Yaskawa INFORM job: DPRINT3D12.JBI

/JOB
//NAME DPRINT3D12
//POS
///NPOS 943,0,0,0,0,0
///TOOL 9
///POSTYPE PULSE
///PULSE
C00000=36380,49514,-121175,76822,-116146,-90921,0
C00001=36311,52030,-113689,77796,-117915,-88696,0
C00002=40966,48656,-123948,71642,-117366,-92253,0
C00003=39960,48244,-125237,72563,-116574,-92522,0
C00004=35348,51596,-114929,78624,-117133,-88953,0
C00005=36233,51994,-113792,77862,-117850,-88717,0
C00006=35618,52329,-112814,78609,-117751,-88361,0
C00007=36492,52745,-111642,77875,-118483,-88119,0
C00008=42195,48620,-124093,70310,-117822,-92440,0
C00009=39827,47660,-127132,72487,-115961,-93077,0
C00010=34247,51723,-114541,79790,-116651,-88720,0
C00011=35148,52115,-113421,79010,-117367,-88487,0
C00012=34913,52339,-112774,79327,-117384,-88271,0
C00013=35382,52553,-112168,78930,-117768,-88145,0
C00014=35564,52380,-112668,78682,-117754,-88312,0
C00015=36124,52085,-113528,78006,-117855,-88627,0
C00016=41195,47951,-126215,71124,-116768,-92950,0
C00017=43098,47003,-129405,68692,-116443,-94111,0
C00018=39318,50776,-117422,74212,-118481,-90143,0
C00019=42795,52637,-112076,71349,-121668,-89077,0
C00020=34867,52594,-112042,79464,-117518,-88051,0
C00021=33535,53991,-108076,81279,-117593,-86746,0
C00022=36088,51585,-114978,77862,-117500,-89049,0
C00023=40156,48632,-124008,72500,-117014,-92178,0
C00024=40156,48569,-124026,72509,-117038,-92154,0
C00025=27110,53258,-109893,66609,-124629,-89161,0
C00026=36380,49453,-121193,76831,-116167,-90898,0
C00027=36311,51973,-113707,77805,-117932,-88673,0
C00028=40967,48594,-123967,71652,-117390,-92229,0
C00029=39960,48181,-125257,72572,-116598,-92498,0
C00030=35348,51539,-114948,78633,-117151,-88931,0
C00031=36233,51937,-113810,77871,-117868,-88695,0
C00032=35619,52272,-112832,78618,-117768,-88339,0
C00033=36492,52688,-111660,77885,-118500,-88098,0
C00034=42195,48557,-124112,70319,-117846,-92417,0
C00035=39828,47596,-127151,72495,-115985,-93052,0
C00036=34247,51665,-114559,79799,-116667,-88698,0
C00037=35149,52058,-113439,79019,-117384,-88465,0
C00038=34914,52282,-112792,79336,-117401,-88249,0
C00039=35382,52497,-112186,78939,-117785,-88123,0
C00040=35565,52323,-112686,78691,-117771,-88290,0
C00041=36125,52027,-113546,78015,-117872,-88605,0
C00042=41195,47887,-126234,71133,-116793,-92926,0
C00043=43079,46945,-129394,68725,-116474,-94076,0
C00044=39319,50717,-117440,74222,-118503,-90120,0
C00045=42764,52562,-112148,71385,-121659,-89066,0
C00046=34867,52538,-112060,79473,-117534,-88029,0
C00047=33548,53922,-108133,81271,-117607,-86737,0
C00048=36088,51527,-114996,77871,-117518,-89026,0
C00049=40156,48569,-124026,72509,-117038,-92154,0
C00050=40157,48507,-124046,72518,-117061,-92130,0
C00051=27147,53215,-109874,66589,-124683,-89138,0
C00052=36381,49392,-121212,76839,-116187,-90874,0
C00053=36312,51915,-113725,77814,-117950,-88651,0
C00054=40967,48531,-123986,71661,-117414,-92206,0
C00055=39961,48118,-125275,72581,-116622,-92474,0
C00056=35348,51481,-114966,78642,-117168,-88908,0
C00057=36234,51879,-113828,77880,-117886,-88673,0
C00058=35619,52216,-112850,78628,-117785,-88317,0
C00059=36492,52632,-111678,77894,-118517,-88076,0
C00060=42195,48495,-124131,70329,-117871,-92394,0
C00061=39828,47531,-127170,72504,-116010,-93028,0
C00062=34248,51608,-114577,79808,-116683,-88676,0
C00063=35149,52001,-113457,79028,-117401,-88442,0
C00064=34914,52225,-112810,79345,-117417,-88227,0
C00065=35382,52440,-112204,78948,-117801,-88101,0
C00066=35565,52266,-112704,78701,-117788,-88268,0
C00067=36125,51970,-113564,78024,-117890,-88583,0
C00068=41196,47823,-126253,71142,-116817,-92902,0
C00069=43061,46888,-129383,68758,-116505,-94040,0
C00070=39319,50658,-117459,74232,-118524,-90097,0
C00071=42733,52486,-112219,71420,-121648,-89055,0
C00072=34868,52481,-112077,79482,-117551,-88007,0
C00073=33561,53853,-108190,81263,-117622,-86728,0
C00074=36088,51469,-115014,77880,-117536,-89004,0
C00075=40157,48507,-124046,72518,-117061,-92130,0
C00076=40157,48444,-124064,72528,-117085,-92106,0
C00077=27184,53173,-109856,66568,-124737,-89114,0
C00078=36381,49332,-121230,76848,-116206,-90851,0
C00079=36312,51858,-113743,77823,-117968,-88629,0
C00080=40968,48469,-124004,71671,-117438,-92182,0
C00081=39961,48055,-125294,72590,-116645,-92450,0
C00082=35349,51423,-114983,78651,-117185,-88885,0
C00083=36234,51822,-113846,77890,-117903,-88650,0
C00084=35619,52159,-112868,78637,-117801,-88295,0
C00085=36493,52576,-111696,77904,-118534,-88054,0
C00086=42196,48432,-124149,70338,-117896,-92370,0
C00087=39828,47467,-127189,72513,-116034,-93003,0
C00088=34248,51550,-114595,79816,-116700,-88653,0
C00089=35150,51944,-113475,79037,-117417,-88420,0
C00090=34914,52168,-112827,79354,-117435,-88204,0
C00091=35383,52383,-112221,78957,-117818,-88079,0
C00092=35565,52209,-112721,78710,-117806,-88246,0
C00093=36125,51913,-113582,78034,-117908,-88561,0
C00094=41196,47759,-126272,71151,-116843,-92878,0
C00095=43042,46831,-129373,68792,-116536,-94005,0
C00096=39320,50599,-117477,74242,-118545,-90075,0
C00097=42701,52411,-112290,71456,-121639,-89045,0
C00098=34868,52424,-112095,79491,-117568,-87985,0
C00099=33573,53785,-108246,81255,-117636,-86720,0
C00100=36089,51411,-115032,77889,-117554,-88982,0
C00101=40157,48444,-124064,72528,-117085,-92106,0
C00102=40157,48382,-124082,72537,-117108,-92083,0
C00103=27222,53130,-109837,66548,-124791,-89091,0
C00104=36381,49271,-121249,76857,-116226,-90827,0
C00105=36312,51801,-113761,77833,-117986,-88607,0
C00106=40968,48407,-124023,71680,-117462,-92159,0
C00107=39962,47992,-125312,72599,-116669,-92426,0
C00108=35349,51365,-115002,78660,-117202,-88863,0
C00109=36234,51765,-113864,77899,-117922,-88628,0
C00110=35620,52102,-112886,78646,-117818,-88272,0
C00111=36493,52519,-111713,77913,-118553,-88032,0
C00112=42196,48370,-124167,70348,-117922,-92347,0
C00113=39829,47402,-127207,72522,-116059,-92979,0
C00114=34248,51492,-114613,79825,-116716,-88631,0
C00115=35150,51887,-113492,79046,-117435,-88398,0
C00116=34915,52111,-112845,79363,-117451,-88182,0
C00117=35383,52327,-112239,78966,-117836,-88057,0
C00118=35566,52153,-112739,78719,-117823,-88224,0
C00119=36126,51856,-113599,78043,-117925,-88538,0
C00120=41196,47695,-126290,71161,-116868,-92854,0
C00121=43024,46774,-129362,68825,-116567,-93970,0
C00122=39320,50540,-117494,74251,-118565,-90053,0
C00123=42670,52335,-112361,71492,-121630,-89034,0
C00124=34868,52368,-112113,79500,-117584,-87963,0
C00125=33586,53716,-108303,81247,-117649,-86710,0
C00126=36089,51353,-115050,77899,-117572,-88959,0
C00127=40157,48382,-124082,72537,-117108,-92083,0
C00128=40158,48319,-124101,72546,-117131,-92059,0
C00129=27259,53088,-109818,66528,-124845,-89067,0
C00130=36382,49210,-121266,76866,-116246,-90804,0
C00131=36313,51744,-113779,77842,-118003,-88585,0
C00132=40968,48344,-124041,71689,-117486,-92135,0
C00133=39962,47928,-125330,72608,-116693,-92402,0
C00134=35350,51307,-115019,78669,-117220,-88840,0
C00135=36235,51707,-113881,77908,-117939,-88606,0
C00136=35620,52045,-112903,78655,-117836,-88250,0
C00137=36493,52463,-111731,77923,-118570,-88010,0
C00138=42197,48307,-124186,70358,-117947,-92323,0
C00139=39829,47338,-127226,72531,-116083,-92955,0
C00140=34248,51435,-114630,79834,-116734,-88608,0
C00141=35150,51830,-113510,79055,-117452,-88375,0
C00142=34915,52055,-112863,79372,-117468,-88160,0
C00143=35383,52270,-112257,78975,-117852,-88035,0
C00144=35566,52096,-112757,78728,-117840,-88201,0
C00145=36126,51799,-113617,78052,-117942,-88516,0
C00146=41197,47632,-126308,71170,-116893,-92830,0
C00147=43005,46717,-129350,68858,-116598,-93934,0
C00148=39320,50481,-117513,74261,-118586,-90030,0
C00149=42639,52260,-112432,71528,-121621,-89023,0
C00150=34868,52311,-112131,79509,-117600,-87941,0
C00151=33599,53647,-108359,81239,-117664,-86702,0
C00152=36089,51296,-115067,77908,-117590,-88936,0
C00153=40158,48319,-124101,72546,-117131,-92059,0
C00154=40158,48257,-124119,72556,-117155,-92035,0
C00155=27296,53046,-109799,66508,-124901,-89043,0
C00156=36382,49149,-121284,76874,-116266,-90780,0
C00157=36313,51687,-113796,77851,-118022,-88563,0
C00158=40969,48282,-124059,71699,-117510,-92111,0
C00159=39963,47865,-125349,72617,-116716,-92378,0
C00160=35350,51250,-115036,78678,-117238,-88817,0
C00161=36235,51650,-113899,77918,-117956,-88584,0
C00162=35620,51988,-112921,78664,-117853,-88228,0
C00163=36494,52407,-111748,77932,-118587,-87988,0
C00164=42197,48245,-124204,70368,-117972,-92300,0
C00165=39830,47274,-127245,72540,-116107,-92930,0
C00166=34249,51377,-114648,79842,-116750,-88585,0
C00167=35150,51773,-113528,79064,-117469,-88353,0
C00168=34915,51998,-112880,79381,-117484,-88137,0
C00169=35384,52214,-112274,78984,-117869,-88013,0
C00170=35566,52039,-112774,78737,-117856,-88179,0
C00171=36126,51742,-113635,78061,-117961,-88494,0
C00172=41197,47568,-126327,71179,-116919,-92806,0
C00173=42987,46660,-129340,68891,-116629,-93899,0
C00174=39321,50422,-117530,74271,-118607,-90007,0
C00175=42608,52184,-112503,71563,-121611,-89012,0
C00176=34869,52255,-112148,79518,-117617,-87919,0
C00177=33612,53578,-108415,81230,-117678,-86693,0
C00178=36090,51238,-115084,77917,-117608,-88914,0
C00179=40158,48257,-124119,72556,-117155,-92035,0
C00180=40159,48194,-124136,72565,-117179,-92011,0
C00181=27333,53003,-109780,66488,-124955,-89020,0
C00182=36383,49088,-121303,76883,-116285,-90756,0
C00183=36313,51629,-113814,77861,-118039,-88540,0
C00184=40969,48219,-124078,71709,-117534,-92087,0
C00185=39963,47802,-125367,72626,-116740,-92354,0
C00186=35350,51192,-115055,78687,-117255,-88795,0
C00187=36235,51593,-113917,77927,-117975,-88561,0
C00188=35621,51931,-112938,78674,-117870,-88206,0
C00189=36494,52350,-111766,77942,-118604,-87967,0
C00190=42198,48182,-124223,70377,-117996,-92276,0
C00191=39830,47209,-127263,72548,-116131,-92905,0
C00192=34249,51320,-114665,79851,-116767,-88563,0
C00193=35151,51716,-113545,79073,-117485,-88331,0
C00194=34916,51941,-112898,79390,-117501,-88115,0
C00195=35384,52157,-112292,78994,-117885,-87990,0
C00196=35567,51982,-112792,78747,-117873,-88157,0
C00197=36127,51685,-113652,78071,-117978,-88472,0
C00198=41198,47504,-126345,71188,-116944,-92782,0
C00199=42968,46603,-129328,68924,-116660,-93863,0
C00200=39321,50364,-117548,74281,-118628,-89985,0
C00201=42577,52108,-112573,71599,-121601,-89001,0
C00202=34869,52199,-112166,79527,-117633,-87896,0
C00203=33624,53509,-108472,81222,-117693,-86684,0
C00204=36090,51180,-115103,77926,-117626,-88891,0
C00205=40159,48194,-124136,72565,-117179,-92011,0
C00206=40159,48132,-124155,72574,-117202,-91987,0
C00207=27370,52961,-109760,66468,-125010,-88996,0
C00208=36383,49027,-121320,76892,-116306,-90732,0
C00209=36314,51572,-113831,77870,-118057,-88518,0
C00210=40970,48157,-124095,71718,-117559,-92063,0
C00211=39963,47739,-125386,72636,-116765,-92330,0
C00212=35351,51134,-115072,78696,-117272,-88772,0
C00213=36236,51536,-113934,77936,-117992,-88539,0
C00214=35621,51875,-112956,78683,-117887,-88184,0
C00215=36494,52294,-111783,77952,-118622,-87945,0
C00216=42198,48120,-124241,70387,-118022,-92253,0
C00217=39831,47145,-127282,72557,-116157,-92880,0
C00218=34250,51262,-114683,79860,-116783,-88540,0
C00219=35151,51659,-113563,79082,-117502,-88308,0
C00220=34916,51884,-112915,79399,-117517,-88093,0
C00221=35384,52101,-112309,79003,-117902,-87968,0
C00222=35567,51926,-112809,78756,-117891,-88135,0
C00223=36127,51628,-113670,78080,-117995,-88449,0
C00224=41198,47440,-126363,71198,-116969,-92758,0
C00225=42950,46547,-129317,68957,-116691,-93828,0
C00226=39321,50305,-117566,74291,-118649,-89962,0
C00227=42546,52033,-112644,71635,-121592,-88990,0
C00228=34869,52142,-112183,79536,-117649,-87874,0
C00229=33637,53440,-108528,81214,-117707,-86675,0
C00230=36090,51122,-115120,77935,-117644,-88869,0
C00231=40159,48132,-124155,72574,-117202,-91987,0
C00232=40160,48070,-124173,72584,-117227,-91964,0
C00233=27407,52919,-109740,66448,-125064,-88972,0
C00234=36383,48966,-121338,76901,-116326,-90708,0
C00235=36314,51515,-113848,77880,-118075,-88495,0
C00236=40970,48095,-124113,71728,-117583,-92040,0
C00237=39964,47676,-125404,72645,-116789,-92305,0
C00238=35351,51077,-115089,78705,-117290,-88749,0
C00239=36236,51479,-113951,77946,-118010,-88517,0
C00240=35621,51818,-112973,78692,-117905,-88161,0
C00241=36495,52238,-111800,77961,-118639,-87923,0
C00242=42198,48057,-124258,70397,-118047,-92229,0
C00243=39831,47081,-127300,72566,-116181,-92856,0
C00244=34250,51205,-114700,79869,-116800,-88517,0
C00245=35151,51602,-113580,79091,-117520,-88286,0
C00246=34916,51828,-112933,79408,-117534,-88071,0
C00247=35385,52044,-112327,79012,-117919,-87946,0
C00248=35567,51869,-112827,78765,-117908,-88112,0
C00249=36127,51570,-113687,78090,-118014,-88427,0
C00250=41198,47377,-126382,71207,-116994,-92734,0
C00251=42932,46490,-129305,68991,-116722,-93793,0
C00252=39322,50246,-117583,74301,-118670,-89940,0
C00253=42514,51957,-112714,71671,-121583,-88979,0
C00254=34870,52086,-112200,79545,-117667,-87852,0
C00255=33650,53371,-108584,81206,-117722,-86666,0
C00256=36091,51065,-115137,77945,-117662,-88846,0
C00257=40160,48070,-124173,72584,-117227,-91964,0
C00258=40160,48007,-124192,72593,-117249,-91940,0
C00259=27444,52877,-109721,66429,-125119,-88948,0
C00260=36384,48906,-121355,76910,-116345,-90684,0
C00261=36314,51458,-113866,77889,-118093,-88473,0
C00262=40970,48032,-124132,71737,-117607,-92016,0
C00263=39964,47613,-125422,72654,-116813,-92281,0
C00264=35351,51019,-115106,78714,-117308,-88727,0
C00265=36236,51421,-113969,77955,-118029,-88494,0
C00266=35622,51761,-112990,78702,-117922,-88139,0
C00267=36495,52182,-111818,77971,-118657,-87901,0
C00268=42199,47995,-124277,70407,-118072,-92206,0
C00269=39831,47016,-127318,72575,-116205,-92831,0
C00270=34250,51147,-114718,79877,-116816,-88494,0
C00271=35152,51545,-113597,79101,-117537,-88263,0
C00272=34917,51771,-112950,79417,-117551,-88049,0
C00273=35385,51988,-112344,79021,-117937,-87924,0
C00274=35568,51812,-112844,78774,-117925,-88090,0
C00275=36128,51513,-113704,78099,-118031,-88405,0
C00276=41199,47313,-126400,71217,-117019,-92709,0
C00277=42913,46433,-129294,69024,-116752,-93757,0
C00278=39322,50187,-117601,74311,-118691,-89917,0
C00279=42483,51882,-112784,71707,-121574,-88968,0
C00280=34870,52029,-112217,79555,-117683,-87830,0
C00281=33663,53302,-108640,81198,-117737,-86657,0
C00282=36091,51007,-115155,77954,-117680,-88823,0
C00283=40160,48007,-124192,72593,-117249,-91940,0
C00284=40160,47945,-124209,72603,-117274,-91915,0
C00285=27481,52836,-109701,66409,-125173,-88925,0
C00286=36384,48845,-121373,76918,-116366,-90660,0
C00287=36315,51401,-113883,77899,-118110,-88451,0
C00288=40971,47970,-124149,71747,-117631,-91992,0
C00289=39965,47549,-125440,72663,-116837,-92257,0
C00290=35351,50961,-115124,78723,-117325,-88704,0
C00291=36237,51364,-113986,77965,-118046,-88472,0
C00292=35622,51704,-113007,78711,-117939,-88117,0
C00293=36495,52125,-111835,77981,-118674,-87878,0
C00294=42199,47932,-124294,70417,-118098,-92182,0
C00295=39832,46952,-127336,72584,-116230,-92807,0
C00296=34250,51090,-114735,79886,-116833,-88472,0
C00297=35152,51488,-113614,79110,-117554,-88241,0
C00298=34917,51714,-112967,79427,-117568,-88026,0
C00299=35385,51931,-112361,79031,-117953,-87902,0
C00300=35568,51756,-112861,78784,-117942,-88068,0
C00301=36128,51456,-113721,78108,-118049,-88382,0
C00302=41199,47249,-126419,71226,-117044,-92685,0
C00303=42895,46377,-129281,69057,-116783,-93721,0
C00304=39323,50128,-117618,74321,-118711,-89894,0
C00305=42452,51806,-112855,71744,-121563,-88957,0
C00306=34870,51973,-112235,79564,-117700,-87807,0
C00307=33675,53233,-108696,81190,-117751,-86648,0
C00308=36091,50949,-115172,77963,-117698,-88801,0
C00309=40160,47945,-124209,72603,-117274,-91915,0
C00310=40161,47882,-124227,72612,-117298,-91892,0
C00311=27518,52794,-109681,66389,-125228,-88901,0
C00312=36384,48784,-121391,76927,-116385,-90636,0
C00313=36315,51344,-113900,77908,-118129,-88428,0
C00314=40971,47908,-124167,71757,-117655,-91968,0
C00315=39965,47486,-125458,72673,-116860,-92233,0
C00316=35352,50904,-115141,78732,-117343,-88682,0
C00317=36237,51307,-114003,77974,-118064,-88449,0
C00318=35622,51648,-113025,78720,-117956,-88094,0
C00319=36496,52069,-111852,77990,-118692,-87856,0
C00320=42200,47870,-124312,70427,-118123,-92158,0
C00321=39832,46888,-127354,72593,-116254,-92782,0
C00322=34251,51032,-114752,79895,-116850,-88449,0
C00323=35152,51431,-113631,79119,-117570,-88219,0
C00324=34917,51658,-112984,79436,-117584,-88003,0
C00325=35386,51875,-112378,79040,-117970,-87880,0
C00326=35568,51699,-112878,78793,-117960,-88046,0
C00327=36128,51399,-113738,78118,-118067,-88360,0
C00328=41200,47185,-126436,71235,-117069,-92660,0
C00329=42876,46320,-129270,69091,-116814,-93685,0
C00330=39323,50069,-117636,74331,-118733,-89871,0
C00331=42420,51731,-112925,71780,-121554,-88945,0
C00332=34871,51916,-112252,79573,-117716,-87785,0
C00333=33688,53165,-108751,81182,-117765,-86638,0
C00334=36092,50892,-115189,77973,-117716,-88778,0
C00335=40161,47882,-124227,72612,-117298,-91892,0
C00336=40161,47820,-124244,72622,-117321,-91868,0
C00337=27555,52752,-109661,66370,-125283,-88877,0
C00338=36385,48723,-121408,76936,-116406,-90612,0
C00339=36315,51287,-113917,77918,-118147,-88406,0
C00340=40972,47845,-124185,71766,-117679,-91944,0
C00341=39965,47423,-125475,72682,-116884,-92208,0
C00342=35352,50846,-115158,78741,-117360,-88658,0
C00343=36237,51250,-114020,77984,-118081,-88427,0
C00344=35623,51591,-113041,78730,-117973,-88072,0
C00345=36496,52013,-111869,78000,-118709,-87834,0
C00346=42200,47807,-124329,70437,-118148,-92134,0
C00347=39833,46824,-127372,72602,-116278,-92757,0
C00348=34251,50975,-114769,79904,-116867,-88426,0
C00349=35153,51374,-113648,79128,-117587,-88196,0
C00350=34918,51601,-113001,79445,-117601,-87981,0
C00351=35386,51819,-112395,79049,-117987,-87857,0
C00352=35569,51643,-112895,78803,-117977,-88023,0
C00353=36129,51342,-113755,78127,-118085,-88337,0
C00354=41200,47122,-126454,71245,-117096,-92636,0
C00355=42858,46264,-129258,69124,-116845,-93650,0
C00356=39323,50011,-117653,74341,-118754,-89848,0
C00357=42389,51655,-112995,71816,-121545,-88934,0
C00358=34871,51860,-112269,79582,-117732,-87762,0
C00359=33701,53096,-108807,81174,-117780,-86629,0
C00360=36092,50834,-115206,77982,-117734,-88755,0
C00361=40161,47820,-124244,72622,-117321,-91868,0
C00362=40162,47758,-124262,72631,-117345,-91843,0
C00363=27592,52710,-109641,66351,-125337,-88853,0
C00364=36385,48663,-121426,76945,-116426,-90588,0
C00365=36316,51230,-113934,77927,-118164,-88383,0
C00366=40972,47783,-124202,71776,-117705,-91921,0
C00367=39966,47360,-125494,72692,-116908,-92184,0
C00368=35352,50788,-115175,78750,-117378,-88636,0
C00369=36238,51193,-114037,77993,-118100,-88404,0
C00370=35623,51534,-113058,78739,-117991,-88050,0
C00371=36496,51957,-111886,78010,-118727,-87812,0
C00372=42201,47745,-124348,70447,-118173,-92110,0
C00373=39833,46759,-127390,72612,-116304,-92732,0
C00374=34251,50917,-114786,79913,-116883,-88403,0
C00375=35153,51317,-113665,79137,-117605,-88173,0
C00376=34918,51544,-113018,79454,-117618,-87959,0
C00377=35386,51762,-112412,79059,-118003,-87835,0
C00378=35569,51586,-112912,78812,-117994,-88001,0
C00379=36129,51286,-113772,78137,-118102,-88315,0
C00380=41201,47058,-126471,71254,-117121,-92612,0
C00381=42840,46207,-129246,69157,-116875,-93614,0
C00382=39324,49952,-117670,74351,-118774,-89825,0
C00383=42357,51579,-113064,71852,-121536,-88922,0
C00384=34871,51804,-112285,79592,-117749,-87740,0
C00385=33714,53027,-108862,81166,-117795,-86620,0
C00386=36093,50776,-115224,77992,-117753,-88733,0
C00387=40162,47758,-124262,72631,-117345,-91843,0
C00388=40162,47695,-124280,72641,-117369,-91820,0
C00389=27629,52669,-109620,66331,-125392,-88830,0
C00390=36385,48602,-121443,76954,-116445,-90565,0
C00391=36316,51173,-113951,77937,-118183,-88361,0
C00392=40972,47721,-124220,71786,-117729,-91897,0
C00393=39966,47297,-125511,72701,-116932,-92160,0
C00394=35353,50731,-115191,78760,-117395,-88613,0
C00395=36238,51136,-114054,78003,-118117,-88382,0
C00396=35623,51478,-113075,78749,-118008,-88027,0
C00397=36497,51901,-111902,78020,-118745,-87790,0
C00398=42201,47683,-124365,70457,-118199,-92087,0
C00399=39833,46695,-127408,72621,-116328,-92707,0
C00400=34252,50860,-114803,79922,-116900,-88380,0
C00401=35153,51260,-113682,79147,-117622,-88151,0
C00402=34918,51488,-113035,79463,-117634,-87936,0
C00403=35387,51706,-112429,79068,-118021,-87812,0
C00404=35569,51529,-112929,78821,-118011,-87978,0
C00405=36129,51229,-113789,78146,-118121,-88292,0
C00406=41201,46995,-126490,71264,-117146,-92587,0
C00407=42821,46151,-129234,69191,-116906,-93578,0
C00408=39324,49893,-117686,74361,-118796,-89803,0
C00409=42326,51504,-113134,71889,-121527,-88911,0
C00410=34872,51748,-112302,79601,-117765,-87718,0
C00411=33726,52958,-108918,81158,-117809,-86611,0
C00412=36093,50719,-115241,78001,-117770,-88709,0
C00413=40162,47695,-124280,72641,-117369,-91820,0
C00414=40162,47633,-124297,72651,-117392,-91795,0
C00415=27666,52627,-109600,66312,-125448,-88806,0
C00416=36386,48541,-121460,76963,-116466,-90540,0
C00417=36316,51116,-113968,77946,-118200,-88338,0
C00418=40973,47658,-124238,71796,-117753,-91872,0
C00419=39967,47234,-125528,72710,-116956,-92135,0
C00420=35353,50673,-115209,78769,-117413,-88590,0
C00421=36238,51079,-114071,78012,-118135,-88359,0
C00422=35624,51421,-113092,78758,-118025,-88004,0
C00423=36497,51845,-111919,78030,-118762,-87768,0
C00424=42201,47620,-124382,70467,-118224,-92063,0
C00425=39834,46631,-127425,72630,-116353,-92683,0
C00426=34252,50803,-114820,79931,-116917,-88357,0
C00427=35154,51203,-113699,79156,-117639,-88128,0
C00428=34919,51431,-113052,79473,-117652,-87913,0
C00429=35387,51650,-112445,79078,-118038,-87790,0
C00430=35570,51473,-112945,78831,-118029,-87956,0
C00431=36130,51172,-113806,78156,-118138,-88270,0
C00432=41201,46931,-126507,71274,-117171,-92563,0
C00433=42803,46095,-129221,69224,-116937,-93542,0
C00434=39324,49834,-117703,74371,-118817,-89779,0
C00435=42294,51428,-113203,71925,-121517,-88899,0
C00436=34872,51691,-112319,79610,-117783,-87696,0
C00437=33739,52889,-108973,81150,-117824,-86601,0
C00438=36093,50661,-115257,78010,-117788,-88687,0
C00439=40162,47633,-124297,72651,-117392,-91795,0
C00440=40163,47571,-124314,72660,-117416,-91771,0
C00441=27702,52586,-109579,66293,-125503,-88781,0
C00442=36386,48481,-121477,76972,-116485,-90516,0
C00443=36317,51059,-113984,77956,-118218,-88315,0
C00444=40973,47596,-124255,71806,-117777,-91849,0
C00445=39967,47171,-125546,72720,-116981,-92110,0
C00446=35353,50616,-115226,78778,-117431,-88567,0
C00447=36239,51022,-114087,78022,-118154,-88336,0
C00448=35624,51365,-113109,78767,-118042,-87982,0
C00449=36497,51789,-111936,78039,-118780,-87746,0
C00450=42202,47558,-124400,70477,-118250,-92039,0
C00451=39834,46567,-127444,72639,-116377,-92658,0
C00452=34252,50745,-114836,79940,-116933,-88334,0
C00453=35154,51146,-113716,79165,-117656,-88105,0
C00454=34919,51374,-113068,79482,-117669,-87891,0
C00455=35387,51593,-112462,79087,-118055,-87768,0
C00456=35570,51416,-112962,78840,-118046,-87934,0
C00457=36130,51115,-113823,78166,-118156,-88247,0
C00458=41202,46867,-126524,71283,-117197,-92539,0
C00459=42785,46039,-129209,69258,-116967,-93506,0
C00460=39325,49776,-117721,74381,-118838,-89757,0
C00461=42263,51353,-113273,71962,-121508,-88888,0
C00462=34872,51635,-112336,79619,-117799,-87673,0
C00463=33752,52820,-109028,81142,-117839,-86592,0
C00464=36094,50604,-115274,78020,-117807,-88664,0
C00465=40163,47571,-124314,72660,-117416,-91771,0
C00466=40163,47509,-124332,72670,-117440,-91747,0
C00467=27739,52545,-109558,66274,-125558,-88758,0
C00468=36387,48420,-121494,76981,-116506,-90492,0
C00469=36317,51002,-114001,77966,-118237,-88293,0
C00470=40974,47534,-124272,71816,-117802,-91824,0
C00471=39967,47108,-125564,72729,-117005,-92086,0
C00472=35354,50558,-115242,78787,-117448,-88544,0
C00473=36239,50965,-114104,78032,-118171,-88314,0
C00474=35624,51308,-113125,78777,-118060,-87960,0
C00475=36498,51733,-111952,78049,-118797,-87724,0
C00476=42202,47496,-124417,70487,-118276,-92015,0
C00477=39835,46503,-127461,72648,-116403,-92633,0
C00478=34253,50688,-114853,79948,-116951,-88311,0
C00479=35154,51090,-113732,79175,-117674,-88083,0
C00480=34919,51318,-113085,79491,-117685,-87868,0
C00481=35388,51537,-112478,79097,-118072,-87745,0
C00482=35570,51360,-112979,78850,-118063,-87911,0
C00483=36130,51058,-113839,78175,-118173,-88224,0
C00484=41202,46804,-126543,71293,-117222,-92514,0
C00485=42766,45983,-129196,69291,-116998,-93471,0
C00486=39325,49717,-117737,74392,-118859,-89734,0
C00487=42232,51277,-113342,71998,-121499,-88876,0
C00488=34873,51579,-112352,79629,-117816,-87650,0
C00489=33765,52751,-109083,81134,-117854,-86583,0
C00490=36094,50546,-115290,78029,-117825,-88641,0
C00491=40163,47509,-124332,72670,-117440,-91747,0
C00492=40164,47446,-124349,72680,-117464,-91723,0
C00493=27776,52503,-109537,66255,-125613,-88734,0
C00494=36387,48359,-121512,76990,-116526,-90468,0
C00495=36317,50945,-114017,77975,-118254,-88270,0
C00496=40974,47472,-124289,71826,-117826,-91801,0
C00497=39968,47045,-125581,72739,-117029,-92062,0
C00498=35354,50501,-115259,78797,-117467,-88521,0
C00499=36239,50908,-114120,78041,-118189,-88291,0
C00500=35625,51252,-113142,78787,-118077,-87937,0
C00501=36498,51677,-111969,78059,-118815,-87701,0
C00502=42203,47434,-124434,70497,-118301,-91991,0
C00503=39835,46439,-127478,72658,-116427,-92607,0
C00504=34253,50631,-114870,79958,-116968,-88288,0
C00505=35155,51033,-113749,79184,-117691,-88060,0
C00506=34920,51261,-113101,79501,-117702,-87845,0
C00507=35388,51481,-112495,79106,-118088,-87723,0
C00508=35570,51303,-112995,78859,-118080,-87888,0
C00509=36131,51001,-113856,78185,-118192,-88202,0
C00510=41203,46740,-126560,71303,-117247,-92489,0
C00511=42748,45927,-129183,69325,-117028,-93435,0
C00512=39325,49658,-117754,74402,-118880,-89710,0
C00513=42200,51202,-113411,72035,-121490,-88864,0
C00514=34873,51523,-112369,79638,-117832,-87628,0
C00515=33778,52683,-109139,81126,-117869,-86573,0
C00516=36094,50489,-115307,78039,-117844,-88618,0
C00517=40164,47446,-124349,72680,-117464,-91723,0
C00518=40164,47384,-124366,72690,-117487,-91698,0
C00519=27813,52462,-109516,66237,-125668,-88710,0
C00520=36387,48299,-121528,77000,-116546,-90444,0
C00521=36318,50888,-114034,77985,-118272,-88248,0
C00522=40975,47410,-124306,71836,-117850,-91776,0
C00523=39968,46982,-125598,72749,-117053,-92037,0
C00524=35355,50443,-115275,78806,-117484,-88498,0
C00525=36240,50851,-114137,78051,-118208,-88268,0
C00526=35625,51195,-113158,78796,-118094,-87914,0
C00527=36498,51621,-111985,78069,-118833,-87679,0
C00528=42203,47371,-124451,70507,-118326,-91968,0
C00529=39836,46374,-127495,72667,-116452,-92582,0
C00530=34253,50573,-114886,79967,-116984,-88265,0
C00531=35155,50976,-113765,79193,-117708,-88037,0
C00532=34920,51205,-113118,79510,-117719,-87823,0
C00533=35388,51425,-112511,79116,-118106,-87700,0
C00534=35571,51247,-113012,78869,-118098,-87866,0
C00535=36131,50944,-113872,78195,-118209,-88179,0
C00536=41203,46677,-126577,71312,-117272,-92465,0
C00537=42730,45870,-129171,69358,-117059,-93399,0
C00538=39326,49600,-117770,74412,-118902,-89688,0
C00539=42168,51126,-113480,72071,-121481,-88852,0
C00540=34873,51467,-112385,79648,-117849,-87606,0
C00541=33790,52614,-109194,81119,-117884,-86564,0
C00542=36095,50431,-115324,78049,-117862,-88595,0
C00543=40164,47384,-124366,72690,-117487,-91698,0
C00544=40164,47322,-124382,72699,-117511,-91674,0
C00545=27850,52421,-109495,66218,-125723,-88686,0
C00546=36388,48238,-121545,77009,-116566,-90419,0
C00547=36318,50831,-114050,77995,-118291,-88225,0
C00548=40975,47348,-124324,71846,-117876,-91752,0
C00549=39969,46919,-125615,72758,-117077,-92012,0
C00550=35355,50386,-115291,78816,-117501,-88475,0
C00551=36240,50794,-114153,78061,-118225,-88245,0
C00552=35625,51139,-113174,78806,-118113,-87892,0
C00553=36499,51565,-112001,78079,-118850,-87656,0
C00554=42204,47309,-124468,70518,-118352,-91943,0
C00555=39836,46310,-127513,72676,-116476,-92557,0
C00556=34254,50516,-114903,79976,-117001,-88242,0
C00557=35155,50919,-113782,79203,-117725,-88014,0
C00558=34920,51148,-113134,79519,-117736,-87800,0
C00559=35389,51368,-112528,79125,-118123,-87678,0
C00560=35571,51191,-113028,78879,-118115,-87843,0
C00561=36131,50887,-113889,78204,-118227,-88156,0
C00562=41204,46613,-126594,71322,-117299,-92440,0
C00563=42712,45814,-129158,69392,-117089,-93363,0
C00564=39326,49541,-117787,74422,-118923,-89665,0
C00565=42137,51051,-113549,72108,-121471,-88841,0
C00566=34874,51410,-112401,79657,-117865,-87583,0
C00567=33803,52545,-109248,81111,-117899,-86554,0
C00568=36095,50374,-115340,78058,-117879,-88572,0
C00569=40164,47322,-124382,72699,-117511,-91674,0
C00570=40165,47260,-124400,72709,-117536,-91650,0
C00571=27886,52380,-109474,66199,-125779,-88662,0
C00572=36388,48178,-121561,77018,-116586,-90395,0
C00573=36318,50774,-114067,78005,-118309,-88202,0
C00574=40975,47285,-124340,71856,-117900,-91728,0
C00575=39969,46856,-125631,72768,-117101,-91987,0
C00576=35355,50328,-115309,78825,-117520,-88452,0
C00577=36240,50737,-114170,78070,-118244,-88223,0
C00578=35626,51082,-113191,78815,-118130,-87869,0
C00579=36499,51509,-112018,78089,-118868,-87634,0
C00580=42204,47247,-124486,70528,-118377,-91919,0
C00581=39836,46246,-127530,72686,-116501,-92532,0
C00582=34254,50459,-114919,79985,-117019,-88219,0
C00583=35156,50862,-113798,79212,-117742,-87992,0
C00584=34920,51092,-113150,79529,-117753,-87778,0
C00585=35389,51312,-112544,79135,-118140,-87655,0
C00586=35572,51134,-113044,78888,-118132,-87820,0
C00587=36132,50831,-113905,78214,-118245,-88134,0
C00588=41204,46550,-126612,71332,-117324,-92416,0
C00589=42693,45759,-129146,69425,-117120,-93327,0
C00590=39327,49482,-117803,74433,-118944,-89641,0
C00591=42105,50975,-113617,72145,-121462,-88828,0
C00592=34874,51354,-112418,79666,-117883,-87560,0
C00593=33816,52476,-109303,81103,-117914,-86544,0
C00594=36095,50316,-115357,78068,-117898,-88549,0
C00595=40165,47260,-124400,72709,-117536,-91650,0
C00596=40165,47198,-124417,72719,-117560,-91625,0
C00597=27923,52339,-109452,66181,-125835,-88638,0
C00598=36388,48117,-121578,77027,-116607,-90371,0
C00599=36319,50718,-114083,78015,-118326,-88179,0
C00600=40976,47223,-124357,71866,-117924,-91704,0
C00601=39969,46794,-125649,72778,-117125,-91963,0
C00602=35355,50271,-115325,78834,-117537,-88429,0
C00603=36241,50680,-114186,78080,-118262,-88200,0
C00604=35626,51026,-113207,78825,-118147,-87847,0
C00605=36499,51453,-112034,78099,-118886,-87612,0
C00606=42204,47185,-124502,70538,-118403,-91896,0
C00607=39837,46182,-127547,72695,-116527,-92507,0
C00608=34254,50402,-114935,79994,-117035,-88196,0
C00609=35156,50806,-113814,79222,-117760,-87968,0
C00610=34921,51036,-113166,79538,-117770,-87755,0
C00611=35389,51256,-112560,79145,-118157,-87632,0
C00612=35572,51078,-113060,78898,-118149,-87798,0
C00613=36132,50774,-113921,78224,-118263,-88111,0
C00614=41204,46486,-126629,71342,-117349,-92391,0
C00615=42675,45703,-129133,69459,-117150,-93291,0
C00616=39327,49424,-117819,74443,-118965,-89618,0
C00617=42073,50899,-113686,72182,-121453,-88817,0
C00618=34874,51298,-112434,79676,-117899,-87538,0
C00619=33829,52407,-109358,81095,-117929,-86535,0
C00620=36096,50259,-115373,78077,-117916,-88526,0
C00621=40165,47198,-124417,72719,-117560,-91625,0
C00622=40166,47136,-124433,72729,-117584,-91601,0
C00623=27960,52298,-109431,66163,-125890,-88614,0
C00624=36389,48057,-121594,77036,-116627,-90346,0
C00625=36319,50661,-114099,78024,-118345,-88156,0
C00626=40976,47161,-124373,71876,-117949,-91679,0
C00627=39970,46731,-125666,72787,-117151,-91938,0
C00628=35356,50214,-115341,78844,-117555,-88405,0
C00629=36241,50624,-114202,78090,-118280,-88177,0
C00630=35626,50969,-113223,78835,-118164,-87823,0
C00631=36500,51397,-112050,78109,-118903,-87589,0
C00632=42205,47122,-124519,70548,-118429,-91871,0
C00633=39837,46118,-127564,72705,-116551,-92482,0
C00634=34255,50344,-114951,80003,-117052,-88173,0
C00635=35156,50749,-113830,79231,-117777,-87946,0
C00636=34921,50979,-113183,79548,-117786,-87732,0
C00637=35390,51200,-112576,79154,-118175,-87610,0
C00638=35572,51022,-113076,78908,-118167,-87775,0
C00639=36132,50717,-113937,78234,-118280,-88088,0
C00640=41205,46423,-126645,71352,-117375,-92366,0
C00641=42657,45647,-129119,69492,-117181,-93255,0
C00642=39327,49365,-117837,74453,-118986,-89595,0
C00643=42042,50824,-113754,72218,-121445,-88805,0
C00644=34875,51242,-112450,79685,-117916,-87515,0
C00645=33842,52338,-109412,81087,-117944,-86525,0
C00646=36096,50201,-115389,78087,-117934,-88503,0
C00647=40166,47136,-124433,72729,-117584,-91601,0
C00648=40166,47073,-124450,72739,-117608,-91577,0
C00649=27996,52257,-109409,66144,-125945,-88590,0
C00650=36389,47996,-121612,77046,-116647,-90322,0
C00651=36319,50604,-114115,78034,-118363,-88133,0
C00652=40977,47099,-124390,71886,-117973,-91655,0
C00653=39970,46668,-125683,72797,-117175,-91914,0
C00654=35356,50156,-115357,78853,-117572,-88382,0
C00655=36241,50567,-114218,78100,-118298,-88154,0
C00656=35626,50913,-113239,78844,-118181,-87801,0
C00657=36500,51341,-112066,78119,-118920,-87567,0
C00658=42205,47060,-124535,70559,-118454,-91848,0
C00659=39838,46054,-127582,72714,-116576,-92456,0
C00660=34255,50287,-114967,80012,-117069,-88149,0
C00661=35157,50692,-113846,79241,-117794,-87923,0
C00662=34921,50923,-113198,79557,-117803,-87709,0
C00663=35390,51144,-112592,79164,-118191,-87587,0
C00664=35572,50965,-113092,78917,-118184,-87753,0
C00665=36133,50660,-113953,78243,-118299,-88065,0
C00666=41205,46359,-126662,71361,-117401,-92341,0
C00667=42639,45591,-129106,69526,-117210,-93219,0
C00668=39328,49307,-117853,74464,-119008,-89572,0
C00669=42010,50748,-113823,72255,-121436,-88792,0
C00670=34875,51186,-112466,79695,-117932,-87493,0
C00671=33855,52269,-109467,81079,-117959,-86515,0
C00672=36096,50144,-115405,78097,-117953,-88480,0
C00673=40166,47073,-124450,72739,-117608,-91577,0
C00674=40167,47011,-124466,72749,-117632,-91552,0
C00675=28033,52216,-109387,66126,-126001,-88566,0
C00676=36389,47936,-121628,77055,-116667,-90298,0
C00677=36320,50547,-114131,78044,-118381,-88111,0
C00678=40977,47037,-124406,71896,-117999,-91631,0
C00679=39971,46605,-125699,72807,-117199,-91889,0
C00680=35356,50099,-115373,78863,-117591,-88359,0
C00681=36242,50510,-114234,78110,-118316,-88131,0
C00682=35627,50857,-113255,78854,-118199,-87778,0
C00683=36500,51285,-112082,78129,-118939,-87544,0
C00684=42206,46998,-124552,70569,-118479,-91823,0
C00685=39838,45990,-127599,72724,-116600,-92431,0
C00686=34255,50230,-114983,80021,-117085,-88126,0
C00687=35157,50636,-113862,79250,-117811,-87900,0
C00688=34922,50866,-113214,79566,-117821,-87686,0
C00689=35390,51088,-112608,79174,-118208,-87565,0
C00690=35573,50909,-113108,78927,-118201,-87729,0
C00691=36133,50604,-113969,78253,-118317,-88042,0
C00692=41206,46296,-126679,71371,-117426,-92316,0
C00693=42621,45536,-129093,69560,-117241,-93183,0
C00694=39328,49248,-117869,74474,-119028,-89548,0
C00695=41978,50673,-113891,72292,-121427,-88780,0
C00696=34875,51130,-112482,79704,-117949,-87470,0
C00697=33867,52201,-109521,81072,-117975,-86506,0
C00698=36097,50087,-115421,78106,-117971,-88456,0
C00699=40167,47011,-124466,72749,-117632,-91552,0
C00700=40167,46949,-124483,72759,-117656,-91527,0
C00701=28070,52176,-109365,66108,-126057,-88542,0
C00702=36390,47875,-121644,77064,-116688,-90273,0
C00703=36320,50490,-114147,78054,-118399,-88088,0
C00704=40977,46975,-124424,71906,-118023,-91607,0
C00705=39971,46542,-125716,72816,-117223,-91864,0
C00706=35357,50042,-115389,78872,-117608,-88336,0
C00707=36242,50453,-114250,78120,-118334,-88108,0
C00708=35627,50800,-113271,78864,-118216,-87755,0
C00709=36501,51229,-112097,78139,-118956,-87522,0
C00710=42206,46936,-124568,70580,-118506,-91799,0
C00711=39838,45926,-127615,72733,-116625,-92406,0
C00712=34256,50173,-114999,80030,-117102,-88102,0
C00713=35157,50579,-113878,79260,-117829,-87877,0
C00714=34922,50810,-113230,79576,-117838,-87663,0
C00715=35390,51032,-112624,79183,-118225,-87542,0
C00716=35573,50853,-113124,78937,-118218,-87707,0
C00717=36133,50547,-113985,78263,-118334,-88019,0
C00718=41206,46232,-126696,71381,-117452,-92292,0
C00719=42602,45480,-129079,69593,-117271,-93147,0
C00720=39328,49190,-117885,74485,-119050,-89525,0
C00721=41946,50597,-113959,72329,-121417,-88768,0
C00722=34875,51074,-112498,79714,-117965,-87447,0
C00723=33880,52132,-109576,81064,-117990,-86496,0
C00724=36097,50029,-115437,78116,-117990,-88433,0
C00725=40167,46949,-124483,72759,-117656,-91527,0
C00726=40167,46887,-124500,72769,-117679,-91503,0
C00727=28106,52135,-109343,66090,-126112,-88518,0
C00728=36390,47815,-121660,77074,-116708,-90249,0
C00729=36320,50434,-114163,78064,-118417,-88065,0
C00730=40978,46913,-124440,71916,-118047,-91582,0
C00731=39972,46479,-125733,72826,-117247,-91839,0
C00732=35357,49984,-115404,78882,-117626,-88313,0
C00733=36242,50396,-114266,78129,-118353,-88085,0
C00734=35628,50744,-113287,78874,-118234,-87732,0
C00735=36501,51173,-112113,78149,-118974,-87499,0
C00736=42206,46874,-124585,70590,-118531,-91775,0
C00737=39839,45862,-127632,72743,-116651,-92381,0
C00738=34256,50116,-115016,80040,-117120,-88079,0
C00739=35158,50523,-113894,79269,-117846,-87854,0
C00740=34922,50754,-113246,79586,-117854,-87641,0
C00741=35391,50976,-112640,79193,-118242,-87519,0
C00742=35573,50796,-113140,78947,-118235,-87684,0
C00743=36134,50490,-114001,78273,-118353,-87996,0
C00744=41207,46169,-126713,71391,-117478,-92267,0
C00745=42584,45425,-129065,69627,-117301,-93111,0
C00746=39329,49131,-117901,74495,-119072,-89502,0
C00747=41914,50522,-114027,72366,-121408,-88755,0
C00748=34876,51018,-112513,79723,-117983,-87424,0
C00749=33893,52063,-109630,81056,-118004,-86486,0
C00750=36097,49972,-115452,78126,-118008,-88410,0
C00751=40167,46887,-124500,72769,-117679,-91503,0
C00752=40168,46825,-124516,72779,-117703,-91478,0
C00753=28143,52095,-109320,66072,-126168,-88494,0
C00754=36391,47754,-121676,77083,-116728,-90225,0
C00755=36321,50377,-114178,78074,-118435,-88042,0
C00756=40978,46851,-124456,71927,-118072,-91558,0
C00757=39972,46417,-125749,72836,-117271,-91814,0
C00758=35357,49927,-115420,78891,-117644,-88289,0
C00759=36243,50340,-114281,78139,-118370,-88062,0
C00760=35628,50687,-113302,78883,-118252,-87710,0
C00761=36501,51118,-112129,78160,-118992,-87476,0
C00762=42207,46812,-124602,70601,-118556,-91751,0
C00763=39839,45798,-127648,72752,-116676,-92355,0
C00764=34256,50059,-115030,80049,-117137,-88056,0
C00765=35158,50466,-113910,79279,-117863,-87831,0
C00766=34923,50698,-113262,79595,-117871,-87617,0
C00767=35391,50920,-112655,79203,-118260,-87496,0
C00768=35574,50740,-113156,78956,-118254,-87661,0
C00769=36134,50434,-114017,78283,-118371,-87974,0
C00770=41207,46105,-126729,71401,-117503,-92242,0
C00771=42566,45369,-129052,69661,-117331,-93075,0
C00772=39329,49073,-117917,74506,-119093,-89479,0
C00773=41882,50446,-114095,72404,-121400,-88743,0
C00774=34876,50962,-112529,79733,-118000,-87402,0
C00775=33906,51994,-109684,81048,-118021,-86476,0
C00776=36098,49915,-115468,78136,-118026,-88387,0
C00777=40168,46825,-124516,72779,-117703,-91478,0
C00778=40168,46763,-124532,72789,-117728,-91454,0
C00779=28179,52054,-109298,66054,-126224,-88470,0
C00780=36391,47694,-121692,77092,-116748,-90200,0
C00781=36321,50320,-114194,78084,-118454,-88019,0
C00782=40979,46789,-124472,71937,-118096,-91533,0
C00783=39972,46354,-125765,72846,-117297,-91789,0
C00784=35358,49870,-115436,78901,-117662,-88266,0
C00785=36243,50283,-114297,78149,-118388,-88039,0
C00786=35628,50631,-113318,78893,-118269,-87686,0
C00787=36502,51062,-112144,78170,-119010,-87454,0
C00788=42207,46750,-124618,70611,-118583,-91726,0
C00789=39840,45734,-127665,72762,-116700,-92330,0
C00790=34257,50002,-115047,80058,-117153,-88033,0
C00791=35158,50409,-113925,79289,-117880,-87808,0
C00792=34923,50641,-113277,79605,-117888,-87595,0
C00793=35391,50864,-112671,79213,-118277,-87473,0
C00794=35574,50684,-113171,78966,-118271,-87638,0
C00795=36134,50377,-114032,78293,-118388,-87950,0
C00796=41207,46042,-126745,71411,-117529,-92217,0
C00797=42548,45314,-129039,69694,-117362,-93038,0
C00798=39330,49014,-117932,74516,-119115,-89456,0
C00799=41850,50371,-114162,72441,-121391,-88731,0
C00800=34876,50906,-112545,79743,-118016,-87378,0
C00801=33919,51925,-109738,81041,-118036,-86466,0
C00802=36098,49858,-115484,78146,-118045,-88364,0
C00803=40168,46763,-124532,72789,-117728,-91454,0
C00804=40168,46701,-124548,72799,-117752,-91429,0
C00805=28216,52014,-109275,66036,-126280,-88446,0
C00806=36391,47634,-121708,77102,-116769,-90175,0
C00807=36321,50264,-114210,78094,-118472,-87996,0
C00808=40979,46727,-124489,71947,-118122,-91509,0
C00809=39973,46291,-125782,72856,-117321,-91764,0
C00810=35358,49813,-115451,78911,-117679,-88242,0
C00811=36243,50226,-114313,78159,-118407,-88016,0
C00812=35628,50575,-113333,78903,-118286,-87664,0
C00813=36502,51006,-112160,78180,-119027,-87431,0
C00814=42208,46688,-124634,70622,-118608,-91702,0
C00815=39840,45670,-127682,72772,-116725,-92304,0
C00816=34257,49945,-115063,80067,-117170,-88009,0
C00817=35159,50353,-113941,79298,-117898,-87784,0
C00818=34923,50585,-113293,79614,-117906,-87572,0
C00819=35392,50808,-112686,79222,-118294,-87451,0
C00820=35574,50628,-113187,78976,-118288,-87615,0
C00821=36135,50321,-114048,78303,-118407,-87927,0
C00822=41208,45979,-126762,71421,-117555,-92192,0
C00823=42530,45259,-129025,69728,-117392,-93002,0
C00824=39330,48956,-117948,74527,-119135,-89432,0
C00825=41819,50295,-114230,72478,-121382,-88718,0
C00826=34877,50850,-112560,79752,-118033,-87356,0
C00827=33932,51856,-109792,81033,-118050,-86456,0
C00828=36098,49800,-115499,78155,-118063,-88340,0
C00829=40168,46701,-124548,72799,-117752,-91429,0
C00830=40169,46639,-124564,72809,-117776,-91404,0
C00831=28253,51974,-109252,66019,-126336,-88422,0
C00832=36392,47573,-121724,77111,-116790,-90151,0
C00833=36322,50207,-114225,78104,-118491,-87972,0
C00834=40979,46665,-124505,71958,-118147,-91484,0
C00835=39973,46228,-125798,72866,-117345,-91739,0
C00836=35358,49756,-115467,78920,-117698,-88219,0
C00837=36244,50170,-114328,78169,-118425,-87993,0
C00838=35629,50519,-113349,78913,-118304,-87641,0
C00839=36502,50950,-112175,78190,-119046,-87408,0
C00840=42208,46626,-124650,70632,-118634,-91677,0
C00841=39841,45606,-127698,72781,-116751,-92279,0
C00842=34257,49888,-115078,80077,-117187,-87986,0
C00843=35159,50296,-113956,79308,-117915,-87761,0
C00844=34924,50529,-113308,79624,-117923,-87548,0
C00845=35392,50752,-112702,79232,-118311,-87428,0
C00846=35575,50571,-113202,78986,-118306,-87592,0
C00847=36135,50264,-114063,78313,-118425,-87905,0
C00848=41208,45915,-126778,71432,-117580,-92167,0
C00849=42512,45203,-129010,69762,-117422,-92966,0
C00850=39330,48897,-117964,74537,-119157,-89409,0
C00851=41786,50219,-114297,72516,-121373,-88705,0
C00852=34877,50794,-112575,79762,-118049,-87333,0
C00853=33945,51787,-109845,81025,-118067,-86446,0
C00854=36099,49743,-115515,78165,-118081,-88317,0
C00855=40169,46639,-124564,72809,-117776,-91404,0
C00856=40169,46577,-124580,72819,-117801,-91380,0
C00857=28289,51933,-109230,66001,-126392,-88397,0
C00858=36392,47513,-121740,77121,-116809,-90126,0
C00859=36322,50151,-114240,78114,-118508,-87950,0
C00860=40980,46603,-124520,71968,-118171,-91460,0
C00861=39974,46166,-125814,72876,-117370,-91714,0
C00862=35359,49698,-115482,78930,-117715,-88196,0
C00863=36244,50113,-114344,78179,-118443,-87970,0
C00864=35629,50463,-113364,78923,-118322,-87618,0
C00865=36503,50895,-112191,78200,-119063,-87386,0
C00866=42209,46564,-124666,70643,-118660,-91653,0
C00867=39841,45542,-127714,72791,-116776,-92254,0
C00868=34258,49831,-115094,80086,-117205,-87963,0
C00869=35159,50240,-113972,79318,-117932,-87738,0
C00870=34924,50473,-113324,79634,-117939,-87526,0
C00871=35392,50696,-112717,79242,-118329,-87405,0
C00872=35575,50515,-113218,78996,-118323,-87569,0
C00873=36135,50208,-114079,78323,-118443,-87881,0
C00874=41209,45852,-126794,71442,-117607,-92142,0
C00875=42493,45148,-128996,69796,-117452,-92930,0
C00876=39331,48839,-117979,74548,-119178,-89385,0
C00877=41755,50144,-114365,72553,-121365,-88693,0
C00878=34877,50738,-112591,79772,-118067,-87310,0
C00879=33958,51719,-109899,81018,-118081,-86435,0
C00880=36099,49686,-115530,78175,-118100,-88294,0
C00881=40169,46577,-124580,72819,-117801,-91380,0
C00882=40170,46515,-124596,72830,-117825,-91355,0
C00883=33479,46360,-124926,79808,-114738,-90748,0
C00884=36392,47452,-121755,77130,-116830,-90101,0
C00885=36322,50094,-114256,78124,-118526,-87927,0
C00886=40980,46541,-124536,71978,-118196,-91435,0
C00887=39974,46103,-125830,72886,-117394,-91689,0
C00888=35359,49641,-115498,78940,-117733,-88172,0
C00889=36244,50056,-114359,78189,-118462,-87947,0
C00890=35629,50406,-113379,78933,-118339,-87595,0
C00891=36503,50839,-112206,78211,-119081,-87363,0
C00892=42209,46502,-124682,70654,-118685,-91629,0
C00893=39841,45478,-127730,72801,-116800,-92228,0
C00894=34258,49774,-115109,80095,-117222,-87939,0
C00895=35160,50183,-113987,79327,-117949,-87715,0
C00896=34924,50417,-113339,79643,-117956,-87502,0
C00897=35393,50640,-112732,79252,-118346,-87382,0
C00898=35575,50459,-113233,79006,-118341,-87547,0
C00899=36136,50151,-114094,78333,-118461,-87858,0
C00900=41209,45789,-126810,71452,-117632,-92117,0
C00901=42475,45093,-128982,69829,-117482,-92893,0
C00902=39331,48781,-117995,74559,-119200,-89362,0
C00903=41722,50068,-114432,72590,-121355,-88680,0
C00904=34878,50683,-112606,79782,-118084,-87287,0
C00905=33971,51650,-109953,81010,-118098,-86425,0
C00906=36099,49629,-115546,78185,-118118,-88270,0
C00907=40170,46515,-124596,72830,-117825,-91355,0
C00908=40170,46453,-124612,72840,-117849,-91330,0
C00909=33520,46312,-124902,79779,-114785,-90715,0
C00910=36393,47392,-121771,77140,-116851,-90077,0
C00911=36323,50037,-114271,78134,-118545,-87903,0
C00912=40981,46479,-124552,71989,-118221,-91411,0
C00913=39974,46040,-125846,72896,-117418,-91664,0
C00914=35359,49584,-115513,78949,-117752,-88149,0
C00915=36245,50000,-114374,78199,-118479,-87924,0
C00916=35630,50350,-113395,78943,-118356,-87572,0
C00917=36503,50783,-112221,78221,-119098,-87341,0
C00918=42209,46440,-124697,70664,-118711,-91604,0
C00919=39842,45414,-127746,72811,-116825,-92203,0
C00920=34258,49717,-115124,80105,-117239,-87916,0
C00921=35160,50127,-114002,79337,-117968,-87692,0
C00922=34925,50360,-113354,79653,-117973,-87479,0
C00923=35393,50584,-112748,79262,-118363,-87359,0
C00924=35576,50403,-113248,79016,-118358,-87523,0
C00925=36136,50095,-114109,78343,-118479,-87835,0
C00926=41210,45725,-126827,71462,-117659,-92092,0
C00927=42457,45038,-128967,69863,-117513,-92857,0
C00928=39331,48722,-118010,74569,-119221,-89338,0
C00929=41690,49993,-114499,72628,-121347,-88668,0
C00930=34878,50627,-112621,79791,-118100,-87264,0
C00931=33984,51581,-110006,81002,-118113,-86415,0
C00932=36100,49572,-115561,78195,-118137,-88247,0
C00933=40170,46453,-124612,72840,-117849,-91330,0
C00934=40170,46391,-124628,72850,-117873,-91306,0
C00935=33560,46264,-124876,79750,-114831,-90681,0
C00936=36393,47332,-121786,77149,-116871,-90052,0
C00937=36323,49981,-114286,78144,-118563,-87880,0
C00938=40981,46417,-124568,71999,-118246,-91386,0
C00939=39975,45978,-125861,72906,-117443,-91639,0
C00940=35360,49527,-115528,78959,-117769,-88125,0
C00941=36245,49943,-114389,78210,-118497,-87901,0
C00942=35630,50294,-113410,78953,-118375,-87548,0
//INST
///DATE 2025/02/20 16:20
///COMM Generated using RoboDK
///ATTR SC,RW
///GROUP1 RB1
NOP
MOVL C00000 V=30.0 PL=1
MOVL C00001 V=130.0 PL=1
MOVL C00002 V=60.0 PL=1
MOVL C00003 V=60.0 PL=1
MOVL C00004 V=60.0 PL=1
MOVL C00005 V=60.0 PL=1
MOVL C00006 V=130.0 PL=1
MOVL C00007 V=30.0 PL=1
MOVL C00008 V=30.0 PL=1
MOVL C00009 V=30.0 PL=1
MOVL C00010 V=30.0 PL=1
MOVL C00011 V=30.0 PL=1
MOVL C00012 V=30.0 PL=1
MOVL C00013 V=30.0 PL=1
MOVL C00014 V=30.0 PL=1
MOVL C00015 V=130.0 PL=1
MOVL C00016 V=130.0 PL=1
MOVL C00017 V=30.0 PL=1
MOVL C00018 V=130.0 PL=1
MOVL C00019 V=30.0 PL=1
MOVL C00020 V=130.0 PL=1
MOVL C00021 V=30.0 PL=1
MOVL C00022 V=130.0 PL=1
MOVL C00023 V=20.0 PL=1
MOVL C00024 V=130.0 PL=1
MOVL C00025 V=130.0 PL=1
MOVL C00026 V=30.0 PL=1
MOVL C00027 V=130.0 PL=1
MOVL C00028 V=60.0 PL=1
MOVL C00029 V=60.0 PL=1
MOVL C00030 V=60.0 PL=1
MOVL C00031 V=60.0 PL=1
MOVL C00032 V=130.0 PL=1
MOVL C00033 V=30.0 PL=1
MOVL C00034 V=30.0 PL=1
MOVL C00035 V=30.0 PL=1
MOVL C00036 V=30.0 PL=1
MOVL C00037 V=30.0 PL=1
MOVL C00038 V=30.0 PL=1
MOVL C00039 V=30.0 PL=1
MOVL C00040 V=30.0 PL=1
MOVL C00041 V=130.0 PL=1
MOVL C00042 V=130.0 PL=1
MOVL C00043 V=30.0 PL=1
MOVL C00044 V=130.0 PL=1
MOVL C00045 V=30.0 PL=1
MOVL C00046 V=130.0 PL=1
MOVL C00047 V=30.0 PL=1
MOVL C00048 V=130.0 PL=1
MOVL C00049 V=20.0 PL=1
MOVL C00050 V=130.0 PL=1
MOVL C00051 V=130.0 PL=1
MOVL C00052 V=30.0 PL=1
MOVL C00053 V=130.0 PL=1
MOVL C00054 V=60.0 PL=1
MOVL C00055 V=60.0 PL=1
MOVL C00056 V=60.0 PL=1
MOVL C00057 V=60.0 PL=1
MOVL C00058 V=130.0 PL=1
MOVL C00059 V=30.0 PL=1
MOVL C00060 V=30.0 PL=1
MOVL C00061 V=30.0 PL=1
MOVL C00062 V=30.0 PL=1
MOVL C00063 V=30.0 PL=1
MOVL C00064 V=30.0 PL=1
MOVL C00065 V=30.0 PL=1
MOVL C00066 V=30.0 PL=1
MOVL C00067 V=130.0 PL=1
MOVL C00068 V=130.0 PL=1
MOVL C00069 V=30.0 PL=1
MOVL C00070 V=130.0 PL=1
MOVL C00071 V=30.0 PL=1
MOVL C00072 V=130.0 PL=1
MOVL C00073 V=30.0 PL=1
MOVL C00074 V=130.0 PL=1
MOVL C00075 V=20.0 PL=1
MOVL C00076 V=130.0 PL=1
MOVL C00077 V=130.0 PL=1
MOVL C00078 V=30.0 PL=1
MOVL C00079 V=130.0 PL=1
MOVL C00080 V=60.0 PL=1
MOVL C00081 V=60.0 PL=1
MOVL C00082 V=60.0 PL=1
MOVL C00083 V=60.0 PL=1
MOVL C00084 V=130.0 PL=1
MOVL C00085 V=30.0 PL=1
MOVL C00086 V=30.0 PL=1
MOVL C00087 V=30.0 PL=1
MOVL C00088 V=30.0 PL=1
MOVL C00089 V=30.0 PL=1
MOVL C00090 V=30.0 PL=1
MOVL C00091 V=30.0 PL=1
MOVL C00092 V=30.0 PL=1
MOVL C00093 V=130.0 PL=1
MOVL C00094 V=130.0 PL=1
MOVL C00095 V=30.0 PL=1
MOVL C00096 V=130.0 PL=1
MOVL C00097 V=30.0 PL=1
MOVL C00098 V=130.0 PL=1
MOVL C00099 V=30.0 PL=1
MOVL C00100 V=130.0 PL=1
MOVL C00101 V=20.0 PL=1
MOVL C00102 V=130.0 PL=1
MOVL C00103 V=130.0 PL=1
MOVL C00104 V=30.0 PL=1
MOVL C00105 V=130.0 PL=1
MOVL C00106 V=60.0 PL=1
MOVL C00107 V=60.0 PL=1
MOVL C00108 V=60.0 PL=1
MOVL C00109 V=60.0 PL=1
MOVL C00110 V=130.0 PL=1
MOVL C00111 V=30.0 PL=1
MOVL C00112 V=30.0 PL=1
MOVL C00113 V=30.0 PL=1
MOVL C00114 V=30.0 PL=1
MOVL C00115 V=30.0 PL=1
MOVL C00116 V=30.0 PL=1
MOVL C00117 V=30.0 PL=1
MOVL C00118 V=30.0 PL=1
MOVL C00119 V=130.0 PL=1
MOVL C00120 V=130.0 PL=1
MOVL C00121 V=30.0 PL=1
MOVL C00122 V=130.0 PL=1
MOVL C00123 V=30.0 PL=1
MOVL C00124 V=130.0 PL=1
MOVL C00125 V=30.0 PL=1
MOVL C00126 V=130.0 PL=1
MOVL C00127 V=20.0 PL=1
MOVL C00128 V=130.0 PL=1
MOVL C00129 V=130.0 PL=1
MOVL C00130 V=30.0 PL=1
MOVL C00131 V=130.0 PL=1
MOVL C00132 V=60.0 PL=1
MOVL C00133 V=60.0 PL=1
MOVL C00134 V=60.0 PL=1
MOVL C00135 V=60.0 PL=1
MOVL C00136 V=130.0 PL=1
MOVL C00137 V=30.0 PL=1
MOVL C00138 V=30.0 PL=1
MOVL C00139 V=30.0 PL=1
MOVL C00140 V=30.0 PL=1
MOVL C00141 V=30.0 PL=1
MOVL C00142 V=30.0 PL=1
MOVL C00143 V=30.0 PL=1
MOVL C00144 V=30.0 PL=1
MOVL C00145 V=130.0 PL=1
MOVL C00146 V=130.0 PL=1
MOVL C00147 V=30.0 PL=1
MOVL C00148 V=130.0 PL=1
MOVL C00149 V=30.0 PL=1
MOVL C00150 V=130.0 PL=1
MOVL C00151 V=30.0 PL=1
MOVL C00152 V=130.0 PL=1
MOVL C00153 V=20.0 PL=1
MOVL C00154 V=130.0 PL=1
MOVL C00155 V=130.0 PL=1
MOVL C00156 V=30.0 PL=1
MOVL C00157 V=130.0 PL=1
MOVL C00158 V=60.0 PL=1
MOVL C00159 V=60.0 PL=1
MOVL C00160 V=60.0 PL=1
MOVL C00161 V=60.0 PL=1
MOVL C00162 V=130.0 PL=1
MOVL C00163 V=30.0 PL=1
MOVL C00164 V=30.0 PL=1
MOVL C00165 V=30.0 PL=1
MOVL C00166 V=30.0 PL=1
MOVL C00167 V=30.0 PL=1
MOVL C00168 V=30.0 PL=1
MOVL C00169 V=30.0 PL=1
MOVL C00170 V=30.0 PL=1
MOVL C00171 V=130.0 PL=1
MOVL C00172 V=130.0 PL=1
MOVL C00173 V=30.0 PL=1
MOVL C00174 V=130.0 PL=1
MOVL C00175 V=30.0 PL=1
MOVL C00176 V=130.0 PL=1
MOVL C00177 V=30.0 PL=1
MOVL C00178 V=130.0 PL=1
MOVL C00179 V=20.0 PL=1
MOVL C00180 V=130.0 PL=1
MOVL C00181 V=130.0 PL=1
MOVL C00182 V=30.0 PL=1
MOVL C00183 V=130.0 PL=1
MOVL C00184 V=60.0 PL=1
MOVL C00185 V=60.0 PL=1
MOVL C00186 V=60.0 PL=1
MOVL C00187 V=60.0 PL=1
MOVL C00188 V=130.0 PL=1
MOVL C00189 V=30.0 PL=1
MOVL C00190 V=30.0 PL=1
MOVL C00191 V=30.0 PL=1
MOVL C00192 V=30.0 PL=1
MOVL C00193 V=30.0 PL=1
MOVL C00194 V=30.0 PL=1
MOVL C00195 V=30.0 PL=1
MOVL C00196 V=30.0 PL=1
MOVL C00197 V=130.0 PL=1
MOVL C00198 V=130.0 PL=1
MOVL C00199 V=30.0 PL=1
MOVL C00200 V=130.0 PL=1
MOVL C00201 V=30.0 PL=1
MOVL C00202 V=130.0 PL=1
MOVL C00203 V=30.0 PL=1
MOVL C00204 V=130.0 PL=1
MOVL C00205 V=20.0 PL=1
MOVL C00206 V=130.0 PL=1
MOVL C00207 V=130.0 PL=1
MOVL C00208 V=30.0 PL=1
MOVL C00209 V=130.0 PL=1
MOVL C00210 V=60.0 PL=1
MOVL C00211 V=60.0 PL=1
MOVL C00212 V=60.0 PL=1
MOVL C00213 V=60.0 PL=1
MOVL C00214 V=130.0 PL=1
MOVL C00215 V=30.0 PL=1
MOVL C00216 V=30.0 PL=1
MOVL C00217 V=30.0 PL=1
MOVL C00218 V=30.0 PL=1
MOVL C00219 V=30.0 PL=1
MOVL C00220 V=30.0 PL=1
MOVL C00221 V=30.0 PL=1
MOVL C00222 V=30.0 PL=1
MOVL C00223 V=130.0 PL=1
MOVL C00224 V=130.0 PL=1
MOVL C00225 V=30.0 PL=1
MOVL C00226 V=130.0 PL=1
MOVL C00227 V=30.0 PL=1
MOVL C00228 V=130.0 PL=1
MOVL C00229 V=30.0 PL=1
MOVL C00230 V=130.0 PL=1
MOVL C00231 V=20.0 PL=1
MOVL C00232 V=130.0 PL=1
MOVL C00233 V=130.0 PL=1
MOVL C00234 V=30.0 PL=1
MOVL C00235 V=130.0 PL=1
MOVL C00236 V=60.0 PL=1
MOVL C00237 V=60.0 PL=1
MOVL C00238 V=60.0 PL=1
MOVL C00239 V=60.0 PL=1
MOVL C00240 V=130.0 PL=1
MOVL C00241 V=30.0 PL=1
MOVL C00242 V=30.0 PL=1
MOVL C00243 V=30.0 PL=1
MOVL C00244 V=30.0 PL=1
MOVL C00245 V=30.0 PL=1
MOVL C00246 V=30.0 PL=1
MOVL C00247 V=30.0 PL=1
MOVL C00248 V=30.0 PL=1
MOVL C00249 V=130.0 PL=1
MOVL C00250 V=130.0 PL=1
MOVL C00251 V=30.0 PL=1
MOVL C00252 V=130.0 PL=1
MOVL C00253 V=30.0 PL=1
MOVL C00254 V=130.0 PL=1
MOVL C00255 V=30.0 PL=1
MOVL C00256 V=130.0 PL=1
MOVL C00257 V=20.0 PL=1
MOVL C00258 V=130.0 PL=1
MOVL C00259 V=130.0 PL=1
MOVL C00260 V=30.0 PL=1
MOVL C00261 V=130.0 PL=1
MOVL C00262 V=60.0 PL=1
MOVL C00263 V=60.0 PL=1
MOVL C00264 V=60.0 PL=1
MOVL C00265 V=60.0 PL=1
MOVL C00266 V=130.0 PL=1
MOVL C00267 V=30.0 PL=1
MOVL C00268 V=30.0 PL=1
MOVL C00269 V=30.0 PL=1
MOVL C00270 V=30.0 PL=1
MOVL C00271 V=30.0 PL=1
MOVL C00272 V=30.0 PL=1
MOVL C00273 V=30.0 PL=1
MOVL C00274 V=30.0 PL=1
MOVL C00275 V=130.0 PL=1
MOVL C00276 V=130.0 PL=1
MOVL C00277 V=30.0 PL=1
MOVL C00278 V=130.0 PL=1
MOVL C00279 V=30.0 PL=1
MOVL C00280 V=130.0 PL=1
MOVL C00281 V=30.0 PL=1
MOVL C00282 V=130.0 PL=1
MOVL C00283 V=20.0 PL=1
MOVL C00284 V=130.0 PL=1
MOVL C00285 V=130.0 PL=1
MOVL C00286 V=30.0 PL=1
MOVL C00287 V=130.0 PL=1
MOVL C00288 V=60.0 PL=1
MOVL C00289 V=60.0 PL=1
MOVL C00290 V=60.0 PL=1
MOVL C00291 V=60.0 PL=1
MOVL C00292 V=130.0 PL=1
MOVL C00293 V=30.0 PL=1
MOVL C00294 V=30.0 PL=1
MOVL C00295 V=30.0 PL=1
MOVL C00296 V=30.0 PL=1
MOVL C00297 V=30.0 PL=1
MOVL C00298 V=30.0 PL=1
MOVL C00299 V=30.0 PL=1
MOVL C00300 V=30.0 PL=1
MOVL C00301 V=130.0 PL=1
MOVL C00302 V=130.0 PL=1
MOVL C00303 V=30.0 PL=1
MOVL C00304 V=130.0 PL=1
MOVL C00305 V=30.0 PL=1
MOVL C00306 V=130.0 PL=1
MOVL C00307 V=30.0 PL=1
MOVL C00308 V=130.0 PL=1
MOVL C00309 V=20.0 PL=1
MOVL C00310 V=130.0 PL=1
MOVL C00311 V=130.0 PL=1
MOVL C00312 V=30.0 PL=1
MOVL C00313 V=130.0 PL=1
MOVL C00314 V=60.0 PL=1
MOVL C00315 V=60.0 PL=1
MOVL C00316 V=60.0 PL=1
MOVL C00317 V=60.0 PL=1
MOVL C00318 V=130.0 PL=1
MOVL C00319 V=30.0 PL=1
MOVL C00320 V=30.0 PL=1
MOVL C00321 V=30.0 PL=1
MOVL C00322 V=30.0 PL=1
MOVL C00323 V=30.0 PL=1
MOVL C00324 V=30.0 PL=1
MOVL C00325 V=30.0 PL=1
MOVL C00326 V=30.0 PL=1
MOVL C00327 V=130.0 PL=1
MOVL C00328 V=130.0 PL=1
MOVL C00329 V=30.0 PL=1
MOVL C00330 V=130.0 PL=1
MOVL C00331 V=30.0 PL=1
MOVL C00332 V=130.0 PL=1
MOVL C00333 V=30.0 PL=1
MOVL C00334 V=130.0 PL=1
MOVL C00335 V=20.0 PL=1
MOVL C00336 V=130.0 PL=1
MOVL C00337 V=130.0 PL=1
MOVL C00338 V=30.0 PL=1
MOVL C00339 V=130.0 PL=1
MOVL C00340 V=60.0 PL=1
MOVL C00341 V=60.0 PL=1
MOVL C00342 V=60.0 PL=1
MOVL C00343 V=60.0 PL=1
MOVL C00344 V=130.0 PL=1
MOVL C00345 V=30.0 PL=1
MOVL C00346 V=30.0 PL=1
MOVL C00347 V=30.0 PL=1
MOVL C00348 V=30.0 PL=1
MOVL C00349 V=30.0 PL=1
MOVL C00350 V=30.0 PL=1
MOVL C00351 V=30.0 PL=1
MOVL C00352 V=30.0 PL=1
MOVL C00353 V=130.0 PL=1
MOVL C00354 V=130.0 PL=1
MOVL C00355 V=30.0 PL=1
MOVL C00356 V=130.0 PL=1
MOVL C00357 V=30.0 PL=1
MOVL C00358 V=130.0 PL=1
MOVL C00359 V=30.0 PL=1
MOVL C00360 V=130.0 PL=1
MOVL C00361 V=20.0 PL=1
MOVL C00362 V=130.0 PL=1
MOVL C00363 V=130.0 PL=1
MOVL C00364 V=30.0 PL=1
MOVL C00365 V=130.0 PL=1
MOVL C00366 V=60.0 PL=1
MOVL C00367 V=60.0 PL=1
MOVL C00368 V=60.0 PL=1
MOVL C00369 V=60.0 PL=1
MOVL C00370 V=130.0 PL=1
MOVL C00371 V=30.0 PL=1
MOVL C00372 V=30.0 PL=1
MOVL C00373 V=30.0 PL=1
MOVL C00374 V=30.0 PL=1
MOVL C00375 V=30.0 PL=1
MOVL C00376 V=30.0 PL=1
MOVL C00377 V=30.0 PL=1
MOVL C00378 V=30.0 PL=1
MOVL C00379 V=130.0 PL=1
MOVL C00380 V=130.0 PL=1
MOVL C00381 V=30.0 PL=1
MOVL C00382 V=130.0 PL=1
MOVL C00383 V=30.0 PL=1
MOVL C00384 V=130.0 PL=1
MOVL C00385 V=30.0 PL=1
MOVL C00386 V=130.0 PL=1
MOVL C00387 V=20.0 PL=1
MOVL C00388 V=130.0 PL=1
MOVL C00389 V=130.0 PL=1
MOVL C00390 V=30.0 PL=1
MOVL C00391 V=130.0 PL=1
MOVL C00392 V=60.0 PL=1
MOVL C00393 V=60.0 PL=1
MOVL C00394 V=60.0 PL=1
MOVL C00395 V=60.0 PL=1
MOVL C00396 V=130.0 PL=1
MOVL C00397 V=30.0 PL=1
MOVL C00398 V=30.0 PL=1
MOVL C00399 V=30.0 PL=1
MOVL C00400 V=30.0 PL=1
MOVL C00401 V=30.0 PL=1
MOVL C00402 V=30.0 PL=1
MOVL C00403 V=30.0 PL=1
MOVL C00404 V=30.0 PL=1
MOVL C00405 V=130.0 PL=1
MOVL C00406 V=130.0 PL=1
MOVL C00407 V=30.0 PL=1
MOVL C00408 V=130.0 PL=1
MOVL C00409 V=30.0 PL=1
MOVL C00410 V=130.0 PL=1
MOVL C00411 V=30.0 PL=1
MOVL C00412 V=130.0 PL=1
MOVL C00413 V=20.0 PL=1
MOVL C00414 V=130.0 PL=1
MOVL C00415 V=130.0 PL=1
MOVL C00416 V=30.0 PL=1
MOVL C00417 V=130.0 PL=1
MOVL C00418 V=60.0 PL=1
MOVL C00419 V=60.0 PL=1
MOVL C00420 V=60.0 PL=1
MOVL C00421 V=60.0 PL=1
MOVL C00422 V=130.0 PL=1
MOVL C00423 V=30.0 PL=1
MOVL C00424 V=30.0 PL=1
MOVL C00425 V=30.0 PL=1
MOVL C00426 V=30.0 PL=1
MOVL C00427 V=30.0 PL=1
MOVL C00428 V=30.0 PL=1
MOVL C00429 V=30.0 PL=1
MOVL C00430 V=30.0 PL=1
MOVL C00431 V=130.0 PL=1
MOVL C00432 V=130.0 PL=1
MOVL C00433 V=30.0 PL=1
MOVL C00434 V=130.0 PL=1
MOVL C00435 V=30.0 PL=1
MOVL C00436 V=130.0 PL=1
MOVL C00437 V=30.0 PL=1
MOVL C00438 V=130.0 PL=1
MOVL C00439 V=20.0 PL=1
MOVL C00440 V=130.0 PL=1
MOVL C00441 V=130.0 PL=1
MOVL C00442 V=30.0 PL=1
MOVL C00443 V=130.0 PL=1
MOVL C00444 V=60.0 PL=1
MOVL C00445 V=60.0 PL=1
MOVL C00446 V=60.0 PL=1
MOVL C00447 V=60.0 PL=1
MOVL C00448 V=130.0 PL=1
MOVL C00449 V=30.0 PL=1
MOVL C00450 V=30.0 PL=1
MOVL C00451 V=30.0 PL=1
MOVL C00452 V=30.0 PL=1
MOVL C00453 V=30.0 PL=1
MOVL C00454 V=30.0 PL=1
MOVL C00455 V=30.0 PL=1
MOVL C00456 V=30.0 PL=1
MOVL C00457 V=130.0 PL=1
MOVL C00458 V=130.0 PL=1
MOVL C00459 V=30.0 PL=1
MOVL C00460 V=130.0 PL=1
MOVL C00461 V=30.0 PL=1
MOVL C00462 V=130.0 PL=1
MOVL C00463 V=30.0 PL=1
MOVL C00464 V=130.0 PL=1
MOVL C00465 V=20.0 PL=1
MOVL C00466 V=130.0 PL=1
MOVL C00467 V=130.0 PL=1
MOVL C00468 V=30.0 PL=1
MOVL C00469 V=130.0 PL=1
MOVL C00470 V=60.0 PL=1
MOVL C00471 V=60.0 PL=1
MOVL C00472 V=60.0 PL=1
MOVL C00473 V=60.0 PL=1
MOVL C00474 V=130.0 PL=1
MOVL C00475 V=30.0 PL=1
MOVL C00476 V=30.0 PL=1
MOVL C00477 V=30.0 PL=1
MOVL C00478 V=30.0 PL=1
MOVL C00479 V=30.0 PL=1
MOVL C00480 V=30.0 PL=1
MOVL C00481 V=30.0 PL=1
MOVL C00482 V=30.0 PL=1
MOVL C00483 V=130.0 PL=1
MOVL C00484 V=130.0 PL=1
MOVL C00485 V=30.0 PL=1
MOVL C00486 V=130.0 PL=1
MOVL C00487 V=30.0 PL=1
MOVL C00488 V=130.0 PL=1
MOVL C00489 V=30.0 PL=1
MOVL C00490 V=130.0 PL=1
MOVL C00491 V=20.0 PL=1
MOVL C00492 V=130.0 PL=1
MOVL C00493 V=130.0 PL=1
MOVL C00494 V=30.0 PL=1
MOVL C00495 V=130.0 PL=1
MOVL C00496 V=60.0 PL=1
MOVL C00497 V=60.0 PL=1
MOVL C00498 V=60.0 PL=1
MOVL C00499 V=60.0 PL=1
MOVL C00500 V=130.0 PL=1
MOVL C00501 V=30.0 PL=1
MOVL C00502 V=30.0 PL=1
MOVL C00503 V=30.0 PL=1
MOVL C00504 V=30.0 PL=1
MOVL C00505 V=30.0 PL=1
MOVL C00506 V=30.0 PL=1
MOVL C00507 V=30.0 PL=1
MOVL C00508 V=30.0 PL=1
MOVL C00509 V=130.0 PL=1
MOVL C00510 V=130.0 PL=1
MOVL C00511 V=30.0 PL=1
MOVL C00512 V=130.0 PL=1
MOVL C00513 V=30.0 PL=1
MOVL C00514 V=130.0 PL=1
MOVL C00515 V=30.0 PL=1
MOVL C00516 V=130.0 PL=1
MOVL C00517 V=20.0 PL=1
MOVL C00518 V=130.0 PL=1
MOVL C00519 V=130.0 PL=1
MOVL C00520 V=30.0 PL=1
MOVL C00521 V=130.0 PL=1
MOVL C00522 V=60.0 PL=1
MOVL C00523 V=60.0 PL=1
MOVL C00524 V=60.0 PL=1
MOVL C00525 V=60.0 PL=1
MOVL C00526 V=130.0 PL=1
MOVL C00527 V=30.0 PL=1
MOVL C00528 V=30.0 PL=1
MOVL C00529 V=30.0 PL=1
MOVL C00530 V=30.0 PL=1
MOVL C00531 V=30.0 PL=1
MOVL C00532 V=30.0 PL=1
MOVL C00533 V=30.0 PL=1
MOVL C00534 V=30.0 PL=1
MOVL C00535 V=130.0 PL=1
MOVL C00536 V=130.0 PL=1
MOVL C00537 V=30.0 PL=1
MOVL C00538 V=130.0 PL=1
MOVL C00539 V=30.0 PL=1
MOVL C00540 V=130.0 PL=1
MOVL C00541 V=30.0 PL=1
MOVL C00542 V=130.0 PL=1
MOVL C00543 V=20.0 PL=1
MOVL C00544 V=130.0 PL=1
MOVL C00545 V=130.0 PL=1
MOVL C00546 V=30.0 PL=1
MOVL C00547 V=130.0 PL=1
MOVL C00548 V=60.0 PL=1
MOVL C00549 V=60.0 PL=1
MOVL C00550 V=60.0 PL=1
MOVL C00551 V=60.0 PL=1
MOVL C00552 V=130.0 PL=1
MOVL C00553 V=30.0 PL=1
MOVL C00554 V=30.0 PL=1
MOVL C00555 V=30.0 PL=1
MOVL C00556 V=30.0 PL=1
MOVL C00557 V=30.0 PL=1
MOVL C00558 V=30.0 PL=1
MOVL C00559 V=30.0 PL=1
MOVL C00560 V=30.0 PL=1
MOVL C00561 V=130.0 PL=1
MOVL C00562 V=130.0 PL=1
MOVL C00563 V=30.0 PL=1
MOVL C00564 V=130.0 PL=1
MOVL C00565 V=30.0 PL=1
MOVL C00566 V=130.0 PL=1
MOVL C00567 V=30.0 PL=1
MOVL C00568 V=130.0 PL=1
MOVL C00569 V=20.0 PL=1
MOVL C00570 V=130.0 PL=1
MOVL C00571 V=130.0 PL=1
MOVL C00572 V=30.0 PL=1
MOVL C00573 V=130.0 PL=1
MOVL C00574 V=60.0 PL=1
MOVL C00575 V=60.0 PL=1
MOVL C00576 V=60.0 PL=1
MOVL C00577 V=60.0 PL=1
MOVL C00578 V=130.0 PL=1
MOVL C00579 V=30.0 PL=1
MOVL C00580 V=30.0 PL=1
MOVL C00581 V=30.0 PL=1
MOVL C00582 V=30.0 PL=1
MOVL C00583 V=30.0 PL=1
MOVL C00584 V=30.0 PL=1
MOVL C00585 V=30.0 PL=1
MOVL C00586 V=30.0 PL=1
MOVL C00587 V=130.0 PL=1
MOVL C00588 V=130.0 PL=1
MOVL C00589 V=30.0 PL=1
MOVL C00590 V=130.0 PL=1
MOVL C00591 V=30.0 PL=1
MOVL C00592 V=130.0 PL=1
MOVL C00593 V=30.0 PL=1
MOVL C00594 V=130.0 PL=1
MOVL C00595 V=20.0 PL=1
MOVL C00596 V=130.0 PL=1
MOVL C00597 V=130.0 PL=1
MOVL C00598 V=30.0 PL=1
MOVL C00599 V=130.0 PL=1
MOVL C00600 V=60.0 PL=1
MOVL C00601 V=60.0 PL=1
MOVL C00602 V=60.0 PL=1
MOVL C00603 V=60.0 PL=1
MOVL C00604 V=130.0 PL=1
MOVL C00605 V=30.0 PL=1
MOVL C00606 V=30.0 PL=1
MOVL C00607 V=30.0 PL=1
MOVL C00608 V=30.0 PL=1
MOVL C00609 V=30.0 PL=1
MOVL C00610 V=30.0 PL=1
MOVL C00611 V=30.0 PL=1
MOVL C00612 V=30.0 PL=1
MOVL C00613 V=130.0 PL=1
MOVL C00614 V=130.0 PL=1
MOVL C00615 V=30.0 PL=1
MOVL C00616 V=130.0 PL=1
MOVL C00617 V=30.0 PL=1
MOVL C00618 V=130.0 PL=1
MOVL C00619 V=30.0 PL=1
MOVL C00620 V=130.0 PL=1
MOVL C00621 V=20.0 PL=1
MOVL C00622 V=130.0 PL=1
MOVL C00623 V=130.0 PL=1
MOVL C00624 V=30.0 PL=1
MOVL C00625 V=130.0 PL=1
MOVL C00626 V=60.0 PL=1
MOVL C00627 V=60.0 PL=1
MOVL C00628 V=60.0 PL=1
MOVL C00629 V=60.0 PL=1
MOVL C00630 V=130.0 PL=1
MOVL C00631 V=30.0 PL=1
MOVL C00632 V=30.0 PL=1
MOVL C00633 V=30.0 PL=1
MOVL C00634 V=30.0 PL=1
MOVL C00635 V=30.0 PL=1
MOVL C00636 V=30.0 PL=1
MOVL C00637 V=30.0 PL=1
MOVL C00638 V=30.0 PL=1
MOVL C00639 V=130.0 PL=1
MOVL C00640 V=130.0 PL=1
MOVL C00641 V=30.0 PL=1
MOVL C00642 V=130.0 PL=1
MOVL C00643 V=30.0 PL=1
MOVL C00644 V=130.0 PL=1
MOVL C00645 V=30.0 PL=1
MOVL C00646 V=130.0 PL=1
MOVL C00647 V=20.0 PL=1
MOVL C00648 V=130.0 PL=1
MOVL C00649 V=130.0 PL=1
MOVL C00650 V=30.0 PL=1
MOVL C00651 V=130.0 PL=1
MOVL C00652 V=60.0 PL=1
MOVL C00653 V=60.0 PL=1
MOVL C00654 V=60.0 PL=1
MOVL C00655 V=60.0 PL=1
MOVL C00656 V=130.0 PL=1
MOVL C00657 V=30.0 PL=1
MOVL C00658 V=30.0 PL=1
MOVL C00659 V=30.0 PL=1
MOVL C00660 V=30.0 PL=1
MOVL C00661 V=30.0 PL=1
MOVL C00662 V=30.0 PL=1
MOVL C00663 V=30.0 PL=1
MOVL C00664 V=30.0 PL=1
MOVL C00665 V=130.0 PL=1
MOVL C00666 V=130.0 PL=1
MOVL C00667 V=30.0 PL=1
MOVL C00668 V=130.0 PL=1
MOVL C00669 V=30.0 PL=1
MOVL C00670 V=130.0 PL=1
MOVL C00671 V=30.0 PL=1
MOVL C00672 V=130.0 PL=1
MOVL C00673 V=20.0 PL=1
MOVL C00674 V=130.0 PL=1
MOVL C00675 V=130.0 PL=1
MOVL C00676 V=30.0 PL=1
MOVL C00677 V=130.0 PL=1
MOVL C00678 V=60.0 PL=1
MOVL C00679 V=60.0 PL=1
MOVL C00680 V=60.0 PL=1
MOVL C00681 V=60.0 PL=1
MOVL C00682 V=130.0 PL=1
MOVL C00683 V=30.0 PL=1
MOVL C00684 V=30.0 PL=1
MOVL C00685 V=30.0 PL=1
MOVL C00686 V=30.0 PL=1
MOVL C00687 V=30.0 PL=1
MOVL C00688 V=30.0 PL=1
MOVL C00689 V=30.0 PL=1
MOVL C00690 V=30.0 PL=1
MOVL C00691 V=130.0 PL=1
MOVL C00692 V=130.0 PL=1
MOVL C00693 V=30.0 PL=1
MOVL C00694 V=130.0 PL=1
MOVL C00695 V=30.0 PL=1
MOVL C00696 V=130.0 PL=1
MOVL C00697 V=30.0 PL=1
MOVL C00698 V=130.0 PL=1
MOVL C00699 V=20.0 PL=1
MOVL C00700 V=130.0 PL=1
MOVL C00701 V=130.0 PL=1
MOVL C00702 V=30.0 PL=1
MOVL C00703 V=130.0 PL=1
MOVL C00704 V=60.0 PL=1
MOVL C00705 V=60.0 PL=1
MOVL C00706 V=60.0 PL=1
MOVL C00707 V=60.0 PL=1
MOVL C00708 V=130.0 PL=1
MOVL C00709 V=30.0 PL=1
MOVL C00710 V=30.0 PL=1
MOVL C00711 V=30.0 PL=1
MOVL C00712 V=30.0 PL=1
MOVL C00713 V=30.0 PL=1
MOVL C00714 V=30.0 PL=1
MOVL C00715 V=30.0 PL=1
MOVL C00716 V=30.0 PL=1
MOVL C00717 V=130.0 PL=1
MOVL C00718 V=130.0 PL=1
MOVL C00719 V=30.0 PL=1
MOVL C00720 V=130.0 PL=1
MOVL C00721 V=30.0 PL=1
MOVL C00722 V=130.0 PL=1
MOVL C00723 V=30.0 PL=1
MOVL C00724 V=130.0 PL=1
MOVL C00725 V=20.0 PL=1
MOVL C00726 V=130.0 PL=1
MOVL C00727 V=130.0 PL=1
MOVL C00728 V=30.0 PL=1
MOVL C00729 V=130.0 PL=1
MOVL C00730 V=60.0 PL=1
MOVL C00731 V=60.0 PL=1
MOVL C00732 V=60.0 PL=1
MOVL C00733 V=60.0 PL=1
MOVL C00734 V=130.0 PL=1
MOVL C00735 V=30.0 PL=1
MOVL C00736 V=30.0 PL=1
MOVL C00737 V=30.0 PL=1
MOVL C00738 V=30.0 PL=1
MOVL C00739 V=30.0 PL=1
MOVL C00740 V=30.0 PL=1
MOVL C00741 V=30.0 PL=1
MOVL C00742 V=30.0 PL=1
MOVL C00743 V=130.0 PL=1
MOVL C00744 V=130.0 PL=1
MOVL C00745 V=30.0 PL=1
MOVL C00746 V=130.0 PL=1
MOVL C00747 V=30.0 PL=1
MOVL C00748 V=130.0 PL=1
MOVL C00749 V=30.0 PL=1
MOVL C00750 V=130.0 PL=1
MOVL C00751 V=20.0 PL=1
MOVL C00752 V=130.0 PL=1
MOVL C00753 V=130.0 PL=1
MOVL C00754 V=30.0 PL=1
MOVL C00755 V=130.0 PL=1
MOVL C00756 V=60.0 PL=1
MOVL C00757 V=60.0 PL=1
MOVL C00758 V=60.0 PL=1
MOVL C00759 V=60.0 PL=1
MOVL C00760 V=130.0 PL=1
MOVL C00761 V=30.0 PL=1
MOVL C00762 V=30.0 PL=1
MOVL C00763 V=30.0 PL=1
MOVL C00764 V=30.0 PL=1
MOVL C00765 V=30.0 PL=1
MOVL C00766 V=30.0 PL=1
MOVL C00767 V=30.0 PL=1
MOVL C00768 V=30.0 PL=1
MOVL C00769 V=130.0 PL=1
MOVL C00770 V=130.0 PL=1
MOVL C00771 V=30.0 PL=1
MOVL C00772 V=130.0 PL=1
MOVL C00773 V=30.0 PL=1
MOVL C00774 V=130.0 PL=1
MOVL C00775 V=30.0 PL=1
MOVL C00776 V=130.0 PL=1
MOVL C00777 V=20.0 PL=1
MOVL C00778 V=130.0 PL=1
MOVL C00779 V=130.0 PL=1
MOVL C00780 V=30.0 PL=1
MOVL C00781 V=130.0 PL=1
MOVL C00782 V=60.0 PL=1
MOVL C00783 V=60.0 PL=1
MOVL C00784 V=60.0 PL=1
MOVL C00785 V=60.0 PL=1
MOVL C00786 V=130.0 PL=1
MOVL C00787 V=30.0 PL=1
MOVL C00788 V=30.0 PL=1
MOVL C00789 V=30.0 PL=1
MOVL C00790 V=30.0 PL=1
MOVL C00791 V=30.0 PL=1
MOVL C00792 V=30.0 PL=1
MOVL C00793 V=30.0 PL=1
MOVL C00794 V=30.0 PL=1
MOVL C00795 V=130.0 PL=1
MOVL C00796 V=130.0 PL=1
MOVL C00797 V=30.0 PL=1
MOVL C00798 V=130.0 PL=1
MOVL C00799 V=30.0 PL=1
MOVL C00800 V=130.0 PL=1
MOVL C00801 V=30.0 PL=1
MOVL C00802 V=130.0 PL=1
MOVL C00803 V=20.0 PL=1
MOVL C00804 V=130.0 PL=1
MOVL C00805 V=130.0 PL=1
MOVL C00806 V=30.0 PL=1
MOVL C00807 V=130.0 PL=1
MOVL C00808 V=60.0 PL=1
MOVL C00809 V=60.0 PL=1
MOVL C00810 V=60.0 PL=1
MOVL C00811 V=60.0 PL=1
MOVL C00812 V=130.0 PL=1
MOVL C00813 V=30.0 PL=1
MOVL C00814 V=30.0 PL=1
MOVL C00815 V=30.0 PL=1
MOVL C00816 V=30.0 PL=1
MOVL C00817 V=30.0 PL=1
MOVL C00818 V=30.0 PL=1
MOVL C00819 V=30.0 PL=1
MOVL C00820 V=30.0 PL=1
MOVL C00821 V=130.0 PL=1
MOVL C00822 V=130.0 PL=1
MOVL C00823 V=30.0 PL=1
MOVL C00824 V=130.0 PL=1
MOVL C00825 V=30.0 PL=1
MOVL C00826 V=130.0 PL=1
MOVL C00827 V=30.0 PL=1
MOVL C00828 V=130.0 PL=1
MOVL C00829 V=20.0 PL=1
MOVL C00830 V=130.0 PL=1
MOVL C00831 V=130.0 PL=1
MOVL C00832 V=30.0 PL=1
MOVL C00833 V=130.0 PL=1
MOVL C00834 V=60.0 PL=1
MOVL C00835 V=60.0 PL=1
MOVL C00836 V=60.0 PL=1
MOVL C00837 V=60.0 PL=1
MOVL C00838 V=130.0 PL=1
MOVL C00839 V=30.0 PL=1
MOVL C00840 V=30.0 PL=1
MOVL C00841 V=30.0 PL=1
MOVL C00842 V=30.0 PL=1
MOVL C00843 V=30.0 PL=1
MOVL C00844 V=30.0 PL=1
MOVL C00845 V=30.0 PL=1
MOVL C00846 V=30.0 PL=1
MOVL C00847 V=130.0 PL=1
MOVL C00848 V=130.0 PL=1
MOVL C00849 V=30.0 PL=1
MOVL C00850 V=130.0 PL=1
MOVL C00851 V=30.0 PL=1
MOVL C00852 V=130.0 PL=1
MOVL C00853 V=30.0 PL=1
MOVL C00854 V=130.0 PL=1
MOVL C00855 V=20.0 PL=1
MOVL C00856 V=130.0 PL=1
MOVL C00857 V=130.0 PL=1
MOVL C00858 V=30.0 PL=1
MOVL C00859 V=130.0 PL=1
MOVL C00860 V=60.0 PL=1
MOVL C00861 V=60.0 PL=1
MOVL C00862 V=60.0 PL=1
MOVL C00863 V=60.0 PL=1
MOVL C00864 V=130.0 PL=1
MOVL C00865 V=30.0 PL=1
MOVL C00866 V=30.0 PL=1
MOVL C00867 V=30.0 PL=1
MOVL C00868 V=30.0 PL=1
MOVL C00869 V=30.0 PL=1
MOVL C00870 V=30.0 PL=1
MOVL C00871 V=30.0 PL=1
MOVL C00872 V=30.0 PL=1
MOVL C00873 V=130.0 PL=1
MOVL C00874 V=130.0 PL=1
MOVL C00875 V=30.0 PL=1
MOVL C00876 V=130.0 PL=1
MOVL C00877 V=30.0 PL=1
MOVL C00878 V=130.0 PL=1
MOVL C00879 V=30.0 PL=1
MOVL C00880 V=130.0 PL=1
MOVL C00881 V=20.0 PL=1
MOVL C00882 V=130.0 PL=1
MOVL C00883 V=130.0 PL=1
MOVL C00884 V=30.0 PL=1
MOVL C00885 V=130.0 PL=1
MOVL C00886 V=60.0 PL=1
MOVL C00887 V=60.0 PL=1
MOVL C00888 V=60.0 PL=1
MOVL C00889 V=60.0 PL=1
MOVL C00890 V=130.0 PL=1
MOVL C00891 V=30.0 PL=1
MOVL C00892 V=30.0 PL=1
MOVL C00893 V=30.0 PL=1
MOVL C00894 V=30.0 PL=1
MOVL C00895 V=30.0 PL=1
MOVL C00896 V=30.0 PL=1
MOVL C00897 V=30.0 PL=1
MOVL C00898 V=30.0 PL=1
MOVL C00899 V=130.0 PL=1
MOVL C00900 V=130.0 PL=1
MOVL C00901 V=30.0 PL=1
MOVL C00902 V=130.0 PL=1
MOVL C00903 V=30.0 PL=1
MOVL C00904 V=130.0 PL=1
MOVL C00905 V=30.0 PL=1
MOVL C00906 V=130.0 PL=1
MOVL C00907 V=20.0 PL=1
MOVL C00908 V=130.0 PL=1
MOVL C00909 V=130.0 PL=1
MOVL C00910 V=30.0 PL=1
MOVL C00911 V=130.0 PL=1
MOVL C00912 V=60.0 PL=1
MOVL C00913 V=60.0 PL=1
MOVL C00914 V=60.0 PL=1
MOVL C00915 V=60.0 PL=1
MOVL C00916 V=130.0 PL=1
MOVL C00917 V=30.0 PL=1
MOVL C00918 V=30.0 PL=1
MOVL C00919 V=30.0 PL=1
MOVL C00920 V=30.0 PL=1
MOVL C00921 V=30.0 PL=1
MOVL C00922 V=30.0 PL=1
MOVL C00923 V=30.0 PL=1
MOVL C00924 V=30.0 PL=1
MOVL C00925 V=130.0 PL=1
MOVL C00926 V=130.0 PL=1
MOVL C00927 V=30.0 PL=1
MOVL C00928 V=130.0 PL=1
MOVL C00929 V=30.0 PL=1
MOVL C00930 V=130.0 PL=1
MOVL C00931 V=30.0 PL=1
MOVL C00932 V=130.0 PL=1
MOVL C00933 V=20.0 PL=1
MOVL C00934 V=130.0 PL=1
MOVL C00935 V=130.0 PL=1
MOVL C00936 V=30.0 PL=1
MOVL C00937 V=130.0 PL=1
MOVL C00938 V=60.0 PL=1
MOVL C00939 V=60.0 PL=1
MOVL C00940 V=60.0 PL=1
MOVL C00941 V=60.0 PL=1
MOVL C00942 V=130.0 PL=1
END
